# B&R Automation Studio project vibratorControlWithCurrentController (part 4)

#### brdkUpdate.fun - Exported functions and function blocks
```iecst
FUNCTION_BLOCK brdkUpdateCheck (*Reads the information from an update package.*) (*$GROUP=User,$CAT=User,$GROUPICON=User.png,$CATICON=User.png*)
	VAR_INPUT
		enable : BOOL := FALSE; (*Enables the function block.*)
		pFileDevice : UDINT := 0; (*String pointer for file device. Can be created with brdkFilelibrary.*)
	END_VAR
	VAR_OUTPUT
		updateFolderPath : STRING[255] := ''; (*Path of the update folder.*)
		pipFilePath : STRING[255] := ''; (*Path of the pipconfig.xml file.*)
		artransferFilePath : STRING[255] := ''; (*Filepath to "artransfer.br" file*)
		version : STRING[32] := ''; (*Update version number.*)
		id : STRING[255] := ''; (*Update configuration ID.*)
		artransferFileSize : UDINT := 0; (*Update file "artransfer.br" size in bytes.*)
		status : DINT := ERR_FUB_ENABLE_FALSE; (*Status of the function block.*)
	END_VAR
	VAR
		internal : brdk_update_check_internal_typ; (*Internal variables.*)
	END_VAR
END_FUNCTION_BLOCK

FUNCTION brdkUpdateCmpVersion : DINT (*Can compare two version strings. The version string must comply with Semantic Versioning x.x.x. $RETURN=result/error;1 : new > old- 0 : new = old : -1 new < old.*) (*$GROUP=User,$CAT=User,$GROUPICON=User.png,$CATICON=User.png*)
	VAR_INPUT
		pNewVersion : UDINT := 0; (*String pointer to new version.*)
		pOldVersion : UDINT := 0; (*String pointer to old version.*)
	END_VAR
END_FUNCTION

FUNCTION_BLOCK brdkUpdateDelete (*Deletes an update.*) (*$GROUP=User,$CAT=User,$GROUPICON=User.png,$CATICON=User.png*)
	VAR_INPUT
		enable : BOOL := FALSE; (*Enables the function block.*)
		pFileDevice : UDINT := 0; (*String pointer for file device. Can be created with brdkFilelibrary.*)
	END_VAR
	VAR_OUTPUT
		status : DINT := ERR_FUB_ENABLE_FALSE; (*Status of the function block.*)
	END_VAR
	VAR
		internal : brdk_update_delete_internal_typ; (*Internal variables.*)
	END_VAR
END_FUNCTION_BLOCK

FUNCTION_BLOCK brdkUpdateDistributeFTP (*Distributes an update package to a list of PLC's.*) (*$GROUP=User,$CAT=User,$GROUPICON=User.png,$CATICON=User.png*)
	VAR_INPUT
		enable : BOOL := FALSE; (*Enables the function block.*)
		pFileDevice : UDINT := 0; (*String pointer for file device. Can be created with brdkFilelibrary.*)
		client : ARRAY[0..BRDK_UPDATE_MAX_FTP_CLIENTS] OF brdk_update_dist_ftp_client_typ; (*List of FTP clients that will receive the update.*)
		cmd : brdk_update_dist_ftp_cmd_typ; (*Commands.*)
	END_VAR
	VAR_OUTPUT
		status : DINT := ERR_FUB_ENABLE_FALSE; (*Status of the function block.*)
		ready : BOOL := FALSE; (*Function block ready.*)
		version : STRING[32] := ''; (*Update version number.*)
		id : STRING[255] := ''; (*Update configuration ID.*)
		artransferFileSize : UDINT := 0; (*Update file "artransfer.br" size in bytes.*)
		updatePackagesSent : USINT := 0; (*Amount of update packages sent*)
	END_VAR
	VAR
		internal : brdk_update_dist_ftp_int_typ; (*Internal variables.*)
	END_VAR
END_FUNCTION_BLOCK

FUNCTION_BLOCK brdkUpdateManager (*Manages updates.*) (*$GROUP=User,$CAT=User,$GROUPICON=User.png,$CATICON=User.png*)
	VAR_INPUT
		enable : BOOL := FALSE; (*Enables the function block.*)
		pFileDevice : UDINT := 0; (*String pointer for file device. Can be created with brdkFilelibrary.*)
		cmd : brdk_update_manager_cmd_typ; (*Commands.*)
	END_VAR
	VAR_OUTPUT
		running : brdk_update_manager_run_info_typ; (*Running information.*)
		update : brdk_update_manager_upd_info_typ; (*Update information.*)
		ready : BOOL := FALSE; (*Function block ready.*)
		status : DINT := ERR_FUB_ENABLE_FALSE; (*Status of the function block.*)
	END_VAR
	VAR
		internal : brdk_update_manager_internal_typ; (*Internal variables.*)
	END_VAR
END_FUNCTION_BLOCK
```

#### brdkUpdateCheck.c - Reads the information from an update package.
```c
#include <brdkUpdate_func.h>

void brdkUpdateCheck(struct brdkUpdateCheck* inst) {
	brdk_update_check_internal_typ* this = (brdk_update_check_internal_typ*)&inst->internal;

	if(!inst->enable) {
		inst->status = ERR_FUB_ENABLE_FALSE;
		this->state = 0;
	}
	else {

		switch(this->state) {

			case 0: /* check that all pointers are set */
				inst->status = ERR_FUB_BUSY;
				if(inst->pFileDevice != 0) {
					this->simulation = DiagCpuIsARsim();
					this->brdkFileRead_0.enable 		= false;
					brdkFileRead(&this->brdkFileRead_0);
					this->brdkFileRead_0.enable 		= true;
					this->brdkFileRead_0.pFileDevice 	= inst->pFileDevice;
					this->brdkFileRead_0.pFileName 		= (unsigned long)&BRDK_UPDATE_DEFAULT_FILE_NAME;
					this->brdkFileRead_0.pData 			= (unsigned long)&this->buffer;
					this->brdkFileRead_0.dataLength 	= sizeof(this->buffer);
					this->state 						= 10;
				}
				else {
					inst->status 	= BRDK_UPDATE_POINTER_ERROR;
					this->state 	= 999;
				}
				break;

			case 10: /* wait for file to be read */
				brdkFileRead(&this->brdkFileRead_0);
				switch(this->brdkFileRead_0.status) {

					case ERR_OK:
						/* find Path= */
						if(!brdkStrSubStrSearch((unsigned long)&inst->pipFilePath,(unsigned long)&this->buffer,(unsigned long)&"Path",(unsigned long)&"\"",2,true)) {
							inst->status = BRDK_UPDATE_PIP_FILE_ERROR;
							this->state = 999;
						}
						else {
							this->position = brdkStrSearch((unsigned long)&inst->pipFilePath, (unsigned long)&"/");
							if(this->position < 0) {
								inst->status = BRDK_UPDATE_PIP_FILE_ERROR;
								this->state = 999;
							}
							else {
								brdkStrMemClear((unsigned long)&inst->updateFolderPath,sizeof(inst->updateFolderPath));
								brdkStrMemCpy((unsigned long)&inst->updateFolderPath, (unsigned long)&inst->pipFilePath, this->position);
								if(!this->simulation) {
									this->ArProjectGetPackageInfo_0.Execute = false;
									ArProjectGetPackageInfo(&this->ArProjectGetPackageInfo_0);
									brdkStrCpy((unsigned long)&this->ArProjectGetPackageInfo_0.DeviceName, inst->pFileDevice);
									brdkStrCpy((unsigned long)&this->ArProjectGetPackageInfo_0.FilePath, (unsigned long)&inst->pipFilePath);
									this->ArProjectGetPackageInfo_0.Execute = true;
									this->state 							= 20;
								}
								else {	/* ArProjectGetPackageInfo_0 does not work in simulation :-( we will just read the file our self ;-) */
									this->brdkFileRead_0.enable 		= false;
									brdkFileRead(&this->brdkFileRead_0);
									this->brdkFileRead_0.enable 		= true;
									this->brdkFileRead_0.pFileDevice 	= inst->pFileDevice;
									this->brdkFileRead_0.pFileName 		= (unsigned long)&inst->pipFilePath;
									this->brdkFileRead_0.pData 			= (unsigned long)&this->buffer;
									this->brdkFileRead_0.dataLength 	= sizeof(this->buffer);
									this->state 						= 30;
								}
							}
						}
						break;

					case ERR_FUB_BUSY:
						break;

					default:
						inst->status = this->brdkFileRead_0.status;
						break;
				}
				break;

			case 20: /* read update package info */
				ArProjectGetPackageInfo(&this->ArProjectGetPackageInfo_0);
				if(!this->ArProjectGetPackageInfo_0.Error) {
					if(this->ArProjectGetPackageInfo_0.Done) {
						brdkStrCpy((unsigned long)&inst->id,(unsigned long)&this->ArProjectGetPackageInfo_0.ConfigurationID);
						brdkStrCpy((unsigned long)&inst->version,(unsigned long)&this->ArProjectGetPackageInfo_0.ConfigurationVersion);

						this->FileInfo_0.enable = false;
						FileInfo(&this->FileInfo_0);
						this->FileInfo_0.enable = true;
						this->FileInfo_0.pDevice = inst->pFileDevice;
						brdkStrMemClear((unsigned long)&inst->artransferFilePath,sizeof(inst->artransferFilePath));
						brdkStrMemCpy((unsigned long)&inst->artransferFilePath,(unsigned long)&inst->updateFolderPath,sizeof(inst->updateFolderPath));
						brdkStrCat((unsigned long)&inst->artransferFilePath,(unsigned long)&BRDK_UPDATE_AR_TRANSFER_PATH);
						this->FileInfo_0.pName = (unsigned long)&inst->artransferFilePath;
						this->FileInfo_0.pInfo = (unsigned long)&this->updateFileInfo;
						this->state 	= 25;
					}
				}
				else {
					inst->status = this->ArProjectGetPackageInfo_0.StatusID;
				}
				break;

			case 25: /* Read file size of the binary update file "artransfer.br" */
				FileInfo(&this->FileInfo_0);
				switch(this->FileInfo_0.status){

					case ERR_OK:
						inst->artransferFileSize = this->updateFileInfo.size;
						inst->status = ERR_OK;
						this->state = 100;
						break;

					case ERR_FUB_BUSY:
						break;

					default:
						inst->status = this->FileInfo_0.status;
						break;

				}
				break;

			case 30: /* file open pipconfig.xml NB! only for simulation !!! */
				brdkFileRead(&this->brdkFileRead_0);
				switch(this->brdkFileRead_0.status) {

					case ERR_OK:
						/* find configuration ID e.g. <ConfigId>brdkUpdate_Config1</ConfigId> */
						if(!brdkStrSubStrSearch((unsigned long)&inst->id,(unsigned long)&this->buffer,(unsigned long)&"ConfigId",(unsigned long)&"<",1,true)) {
							inst->status = BRDK_UPDATE_PIP_FILE_ERROR;
							this->state = 999;
						}
						else {
							/* find configuration version e.g. <ConfigVersion>1.0.1</ConfigVersion> */
							if(!brdkStrSubStrSearch((unsigned long)&inst->version,(unsigned long)&this->buffer,(unsigned long)&"ConfigVersion",(unsigned long)&"<",1,true)) {
								inst->status = BRDK_UPDATE_PIP_FILE_ERROR;
								this->state = 999;
							}
							else {
								inst->status 	= ERR_OK;
								this->state 	= 100;
							}
						}
						break;

					case ERR_FUB_BUSY:
						break;

					default:
						inst->status = this->brdkFileRead_0.status;
						break;
				}
				break;

			case 100:
				break;

		}
	}
}
```

#### brdkUpdateCmpVersion.c - Can compare two version strings. The version string must comply with Semantic Versioning x.x.x
```c
#include <brdkUpdate_func.h>

signed long brdkUpdateCmpVersion(unsigned long pNewVersion, unsigned long pOldVersion) {
	unsigned long newIdx = 0, oldIdx = 0, newVal = 0, oldVal = 0, cnt = 0;
	char noZero;
	if(pNewVersion != 0 && pOldVersion != 0) {
		while(cnt < 3) {
			noZero = 0;
			while(((char*)pNewVersion)[newIdx] != 46 && ((char*)pNewVersion)[newIdx] != 0) {	/* look for a . */
				if((((char*)pNewVersion)[newIdx]) > 48) noZero = true;	/* make sure that first char is not a 0 */
				if(noZero) newVal += ((char*)pNewVersion)[newIdx];
				newIdx++;
			}
			newIdx++;
			noZero = 0;
			while(((char*)pOldVersion)[oldIdx] != 46 && ((char*)pOldVersion)[oldIdx] != 0) {	/* look for a . */
				if((((char*)pOldVersion)[oldIdx]) > 48) noZero = true;	/* make sure that first char is not a 0 */
				if(noZero) oldVal += ((char*)pOldVersion)[oldIdx];
				oldIdx++;
			}
			oldIdx++;
			if(newVal > oldVal) return 1;
			else if(newVal < oldVal) return -1;
			newVal = oldVal = 0;
			cnt++;
		}
	}
	else return BRDK_UPDATE_POINTER_ERROR;
	return 0;
}
```

#### brdkUpdateDelete.c - Deletes an update.
```c
#include <brdkUpdate_func.h>

void brdkUpdateDelete(struct brdkUpdateDelete* inst) {
	brdk_update_delete_internal_typ* this = (brdk_update_delete_internal_typ*)&inst->internal;

	if(!inst->enable) {
		inst->status = ERR_FUB_ENABLE_FALSE;
		this->state = 0;
	}
	else {

		switch(this->state) {

			case 0: /* check that all pointers are set */
				inst->status = ERR_FUB_BUSY;
				if(inst->pFileDevice != 0) {
					inst->status 						= ERR_FUB_BUSY;
					this->brdkUpdateCheck_0.enable 		= false;
					brdkUpdateCheck(&this->brdkUpdateCheck_0);
					this->brdkUpdateCheck_0.enable 		= true;
					this->brdkUpdateCheck_0.pFileDevice = inst->pFileDevice;
					this->state 						= 10;
				}
				else {
					inst->status 	= BRDK_UPDATE_POINTER_ERROR;
					this->state 	= 999;
				}
				break;

			case 10:
				brdkUpdateCheck(&this->brdkUpdateCheck_0);
				switch(this->brdkUpdateCheck_0.status) {

					case ERR_OK:
						this->DirDeleteEx_0.enable = false;
						DirDeleteEx(&this->DirDeleteEx_0);
						this->DirDeleteEx_0.enable 	= true;
						this->DirDeleteEx_0.pDevice = inst->pFileDevice;
						this->DirDeleteEx_0.pName 	= (unsigned long)&this->brdkUpdateCheck_0.updateFolderPath;
						this->state 				= 20;
						break;

					case ERR_FUB_BUSY:
						break;

					default:
						inst->status = this->brdkUpdateCheck_0.status;
						break;
				}
				break;

			case 20: /* delete update folder */
				DirDeleteEx(&this->DirDeleteEx_0);
				switch(this->DirDeleteEx_0.status) {

					case ERR_OK:
						this->FileDelete_0.enable = false;
						FileDelete(&this->FileDelete_0);
						this->FileDelete_0.enable 	= true;
						this->FileDelete_0.pDevice 	= inst->pFileDevice;
						this->FileDelete_0.pName 	= (unsigned long)&BRDK_UPDATE_DEFAULT_FILE_NAME;
						this->state 				= 30;
						break;

					case ERR_FUB_BUSY:
						break;

					default:
						inst->status = this->DirDeleteEx_0.status;
						break;

				}
				break;

			case 30: /* delete update file */
				FileDelete(&this->FileDelete_0);
				switch(this->FileDelete_0.status) {

					case ERR_OK:
						inst->status 	= ERR_OK;
						this->state 	= 40;
						break;

					case ERR_FUB_BUSY:
						break;

					default:
						inst->status = this->FileDelete_0.status;
						break;

				}
				break;

			case 40: /* done */
				break;

		}
	}
}
```

#### brdkUpdateDistributeFTP.c - Distributes an update package to a list of PLC's via FTP
```c
#include <brdkUpdate_func.h>

void brdkUpdateDistributeFTP(struct brdkUpdateDistributeFTP* inst) {
	brdk_update_dist_ftp_int_typ* this = (brdk_update_dist_ftp_int_typ*) &inst->internal;

	if(!inst->enable) {
		inst->status = ERR_FUB_ENABLE_FALSE;
		this->state = 0;
	}
	else {
		switch(this->state) {

			case 0: /* check that the file device pointer is set */
				if(inst->pFileDevice != 0) {
					inst->status = ERR_OK;
					inst->ready = true;
					this->state = 100;
				}
				else {
					inst->status 	= BRDK_UPDATE_POINTER_ERROR;
					this->state 	= 999;
				}
				break;

			case 100: /* wait for command */
				if(inst->cmd.distributeUpdate || inst->cmd.checkUpdate) {
					inst->ready 						= false;
					inst->status 						= ERR_FUB_BUSY;
					this->brdkUpdateCheck_0.enable 		= false;
					brdkUpdateCheck(&this->brdkUpdateCheck_0);
					this->brdkUpdateCheck_0.enable 		= true;
					this->brdkUpdateCheck_0.pFileDevice	= inst->pFileDevice;
					this->state 						= 110;
				}
				else if(inst->cmd.deleteUpdate) {
					inst->cmd.deleteUpdate 					= false;
					this->brdkUpdateDelete_0.enable			= false;
					brdkUpdateDelete(&this->brdkUpdateDelete_0);
					this->brdkUpdateDelete_0.enable 		= true;
					this->brdkUpdateDelete_0.pFileDevice 	= inst->pFileDevice;
					this->state 							= 200;
				}
				break;

			case 110: /* wait for update to be read */
				brdkUpdateCheck(&this->brdkUpdateCheck_0);
				switch(this->brdkUpdateCheck_0.status) {

					case ERR_OK:
						brdkStrCpy((unsigned long)&inst->id,(unsigned long)&this->brdkUpdateCheck_0.id);
						brdkStrCpy((unsigned long)&inst->version,(unsigned long)&this->brdkUpdateCheck_0.version);
						inst->artransferFileSize = this->brdkUpdateCheck_0.artransferFileSize;
						if(inst->cmd.checkUpdate) {
							inst->cmd.checkUpdate	= false;
							inst->status 			= ERR_OK;
							inst->ready 			= true;
							this->state 			= 100;
						}
						else if(inst->cmd.distributeUpdate) {
							inst->cmd.distributeUpdate = false;
							this->cIdx = 0;						/* reset client idx */
							inst->updatePackagesSent = 0;		/* reset packages sent */
							if(!brdkStrIsEmpty((unsigned long)&inst->client[this->cIdx].pIPAddress)) {
								brdkStrCpy((unsigned long)&this->paramStr,(unsigned long)&"/PROTOCOL=ftp");
								brdkStrCat((unsigned long)&this->paramStr,(unsigned long)&" /SIP=");
								brdkStrCat((unsigned long)&this->paramStr,inst->client[this->cIdx].pIPAddress);
								if(!brdkStrIsEmpty((unsigned long)&inst->client[this->cIdx].pUser)) {
									brdkStrCat((unsigned long)&this->paramStr,(unsigned long)&" /USER=");
									brdkStrCat((unsigned long)&this->paramStr,inst->client[this->cIdx].pUser);
									if(!brdkStrIsEmpty((unsigned long)&inst->client[this->cIdx].pPassword)) {
										brdkStrCat((unsigned long)&this->paramStr,(unsigned long)&" /PASSWORD=");
										brdkStrCat((unsigned long)&this->paramStr,inst->client[this->cIdx].pPassword);
									}
								}
								this->DevLink_0.enable = false;
								DevLink(&this->DevLink_0);
								this->DevLink_0.enable 	= true;
								this->DevLink_0.pDevice = (unsigned long)&BRDK_UPDATE_FTP_DEVICE_NAME;
								this->DevLink_0.pParam 	= (unsigned long)&this->paramStr;
								this->state 			= 120;
							}
						}
						break;

					case ERR_FUB_BUSY:
						break;

					default:
						inst->status = this->brdkUpdateCheck_0.status;
						if(inst->cmd.errorReset) {
							inst->cmd.errorReset 		= false;
							inst->cmd.distributeUpdate 	= false;
							inst->cmd.checkUpdate 		= false;
							inst->status 				= ERR_OK;
							inst->ready 				= true;
							this->state 				= 100;
						}
						break;
				}
				break;

			case 120: /* create dev link for FTP */
				DevLink(&this->DevLink_0);
				switch(this->DevLink_0.status) {

					case ERR_OK:
						this->DirCopy_0.enable 		= false;
						DirCopy(&this->DirCopy_0);
						this->DirCopy_0.enable 		= true;
						this->DirCopy_0.pSrcDev 	= inst->pFileDevice;
						this->DirCopy_0.pSrcDir 	= (unsigned long)&this->brdkUpdateCheck_0.updateFolderPath;
						this->DirCopy_0.pDestDev 	= this->DevLink_0.pDevice;
						this->DirCopy_0.pDestDir 	= 0;
						this->DirCopy_0.option 		= fiOVERWRITE;
						this->state 				= 130;
						break;

					case ERR_FUB_BUSY:
						break;

					default:
						inst->status 				= this->DevLink_0.status;
						if(inst->cmd.errorReset) {
							inst->cmd.errorReset 	= false;
							inst->status 			= ERR_OK;
							inst->ready 			= true;
							this->state 			= 100;
						}
						break;

				}
				break;

			case 130: /* copy update folder to ftp server */
				DirCopy(&this->DirCopy_0);
				switch(this->DirCopy_0.status) {

					case ERR_OK:
						this->FileCopy_0.enable 	= false;
						FileCopy(&this->FileCopy_0);
						this->FileCopy_0.enable 	= true;
						this->FileCopy_0.pSrcDev 	= this->DirCopy_0.pSrcDev;
						this->FileCopy_0.pSrc 		= (unsigned long)&BRDK_UPDATE_DEFAULT_FILE_NAME;
						this->FileCopy_0.pDestDev 	= this->DirCopy_0.pDestDev;
						this->FileCopy_0.pDest 		= this->FileCopy_0.pSrc;
						this->FileCopy_0.option 	= fiOVERWRITE;
						this->state 				= 140;
						break;

					case ERR_FUB_BUSY:
						break;

					default:
						inst->status 				= this->DirCopy_0.status;
						if(inst->cmd.errorReset) {
							inst->cmd.errorReset 	= false;
							inst->status 			= ERR_OK;
							inst->ready 			= true;
							this->state 			= 100;
						}
						break;

				}
				break;

			case 140: /* copy file */
				FileCopy(&this->FileCopy_0);
				switch(this->FileCopy_0.status) {

					case ERR_OK:
						this->DevUnlink_0.enable 	= false;
						DevUnlink(&this->DevUnlink_0);
						this->DevUnlink_0.enable 	= true;
						this->DevUnlink_0.handle 	= this->DevLink_0.handle;
						this->state 				= 150;
						break;

					case ERR_FUB_BUSY:
						break;

					default:
						inst->status 				= this->FileCopy_0.status;
						if(inst->cmd.errorReset) {
							inst->cmd.errorReset 	= false;
							inst->status 			= ERR_OK;
							inst->ready 			= true;
							this->state 			= 100;
						}
						break;

				}
				break;

			case 150: /* unlink file device */
				DevUnlink(&this->DevUnlink_0);
				switch(this->DevUnlink_0.status) {

					case ERR_OK:
						this->cIdx++;						/* reset client idx */
						inst->updatePackagesSent++;			/* Amount of packages sent	*/
						if(this->cIdx < BRDK_UPDATE_MAX_FTP_CLIENTS) {
							if(!brdkStrIsEmpty((unsigned long)&inst->client[this->cIdx].pIPAddress)) {
								brdkStrCpy((unsigned long)&this->paramStr,(unsigned long)&"/PROTOCOL=ftp");
								brdkStrCat((unsigned long)&this->paramStr,(unsigned long)&" /SIP=");
								brdkStrCat((unsigned long)&this->paramStr,inst->client[this->cIdx].pIPAddress);
								if(!brdkStrIsEmpty((unsigned long)&inst->client[this->cIdx].pUser)) {
									brdkStrCat((unsigned long)&this->paramStr,(unsigned long)&" /USER=");
									brdkStrCat((unsigned long)&this->paramStr,inst->client[this->cIdx].pUser);
									if(!brdkStrIsEmpty((unsigned long)&inst->client[this->cIdx].pPassword)) {
										brdkStrCat((unsigned long)&this->paramStr,(unsigned long)&" /PASSWORD=");
										brdkStrCat((unsigned long)&this->paramStr,inst->client[this->cIdx].pPassword);
									}
								}
								this->DevLink_0.enable = false;
								DevLink(&this->DevLink_0);
								this->DevLink_0.enable 	= true;
								this->DevLink_0.pDevice = (unsigned long)&BRDK_UPDATE_FTP_DEVICE_NAME;
								this->DevLink_0.pParam 	= (unsigned long)&this->paramStr;
								this->state 			= 120;
							}
							else {
								inst->status = ERR_OK;
								inst->ready = true;
								this->state = 100;
							}
						}
						else {
							inst->status = ERR_OK;
							inst->ready = true;
							this->state = 100;
						}
						break;

					case ERR_FUB_BUSY:
						break;

					default:
						inst->status 				= this->DevUnlink_0.status;
						if(inst->cmd.errorReset) {
							inst->cmd.errorReset 	= false;
							inst->status 			= ERR_OK;
							inst->ready 			= true;
							this->state 			= 100;
						}
						break;

				}
				break;

			case 200: /* delete update folder */
				brdkUpdateDelete(&this->brdkUpdateDelete_0);
				switch(this->brdkUpdateDelete_0.status) {

					case ERR_OK:
						inst->id[0] 		= 0;
						inst->version[0] 	= 0;
						inst->status 		= BRDK_UPDATE_NOT_FOUND;
						inst->status 		= ERR_OK;
						inst->ready 		= true;
						this->state 		= 100;
						break;

					case ERR_FUB_BUSY:
						break;

					default:
						inst->status = this->brdkUpdateDelete_0.status;
						if(inst->cmd.errorReset) {
							inst->cmd.errorReset = false;
							inst->status = ERR_OK;
							inst->ready = true;
							this->state = 100;
						}
						break;

				}
				break;

		}

	}
}
```

#### brdkUpdateManager.c - Manages updates.
```c
#include <brdkUpdate_func.h>

void brdkUpdateManager(struct brdkUpdateManager* inst) {
	brdk_update_manager_internal_typ* this = (brdk_update_manager_internal_typ*)&inst->internal;

	if(!inst->enable) {
		inst->status = ERR_FUB_ENABLE_FALSE;
		this->state = 0;
	}
	else {
		switch(this->state) {

			case 0: /* check that the file device pointer is set */
				inst->status = ERR_FUB_BUSY;
				if(inst->pFileDevice != 0) {
					this->ArProjectGetInfo_0.Execute = false;
					ArProjectGetInfo(&this->ArProjectGetInfo_0);
					this->ArProjectGetInfo_0.Execute = true;
					this->state = 10;
				}
				else {
					inst->status 	= BRDK_UPDATE_POINTER_ERROR;
					this->state 	= 999;
				}
				break;

			case 10: /* read the running id and version */
				ArProjectGetInfo(&this->ArProjectGetInfo_0);
				if(!this->ArProjectGetInfo_0.Error) {
					if(this->ArProjectGetInfo_0.Done) {
						brdkStrCpy((unsigned long)&inst->running.id,(unsigned long)&this->ArProjectGetInfo_0.ConfigurationID);
						brdkStrCpy((unsigned long)&inst->running.version,(unsigned long)&this->ArProjectGetInfo_0.ConfigurationVersion);
						inst->status = ERR_OK;
						inst->ready = true;
						this->state = 100;
					}
				}
				else {
					inst->status = this->ArProjectGetInfo_0.StatusID;
					if(inst->cmd.errorReset) {
						inst->cmd.errorReset = false;
						inst->status = ERR_OK;
						inst->ready = true;
						this->state = 100;
					}
				}
				break;

			case 100: /* check for commands */
				if(inst->cmd.checkForUpdate || inst->cmd.update || inst->cmd.updateReboot) {
					inst->ready 						= false;
					inst->status 						= ERR_FUB_BUSY;
					this->brdkUpdateCheck_0.enable 		= false;
					brdkUpdateCheck(&this->brdkUpdateCheck_0);
					this->brdkUpdateCheck_0.enable 		= true;
					this->brdkUpdateCheck_0.pFileDevice = inst->pFileDevice;
					this->state 						= 110;
				}
				else if(inst->cmd.deleteUpdate) {
					inst->cmd.deleteUpdate 					= false;
					this->brdkUpdateDelete_0.enable			= false;
					brdkUpdateDelete(&this->brdkUpdateDelete_0);
					this->brdkUpdateDelete_0.enable 		= true;
					this->brdkUpdateDelete_0.pFileDevice 	= inst->pFileDevice;
					this->state 							= 200;
				}
				break;

			case 110: /* wait for update to be read */
				brdkUpdateCheck(&this->brdkUpdateCheck_0);
				switch(this->brdkUpdateCheck_0.status) {

					case ERR_OK:
						if(inst->cmd.checkForUpdate) {
							inst->cmd.checkForUpdate				= false;
							brdkStrCpy((unsigned long)&inst->update.id,(unsigned long)&this->brdkUpdateCheck_0.id);
							brdkStrCpy((unsigned long)&inst->update.version,(unsigned long)&this->brdkUpdateCheck_0.version);
							inst->update.artransferFileSize = this->brdkUpdateCheck_0.artransferFileSize;
							inst->update.status = BRDK_UPDATE_NOT_FOUND;
							if(brdkStrCmp((unsigned long)&inst->update.id,(unsigned long)&inst->running.id) != 0) inst->update.status = BRDK_UPDATE_NO_ID_MATCH;
							this->versionCmp = brdkUpdateCmpVersion((unsigned long)&inst->update.version,(unsigned long)&inst->running.version);
							if(inst->update.status != BRDK_UPDATE_NO_ID_MATCH) {
								if(this->versionCmp > 0) inst->update.status = BRDK_UPDATE_VERSION_NEW_GREATER;
								else if(this->versionCmp < 0) inst->update.status = BRDK_UPDATE_VERSION_NEW_SMALLER;
								else inst->update.status = BRDK_UPDATE_VERSIONS_EQUAL;
							}
							inst->status 	= ERR_OK;
							inst->ready 	= true;
							this->state 	= 100;
						}
						else if(inst->cmd.update || inst->cmd.updateReboot) {
							inst->cmd.update 						= false;
							this->ArProjectInstallPackage_0.Execute = false;
							ArProjectInstallPackage(&this->ArProjectInstallPackage_0);
							this->ArProjectInstallPackage_0.Execute = true;
							brdkStrCpy((unsigned long)&this->ArProjectInstallPackage_0.DeviceName, inst->pFileDevice);
							brdkStrCpy((unsigned long)&this->ArProjectInstallPackage_0.FilePath, (unsigned long)&this->brdkUpdateCheck_0.pipFilePath);
							this->state 							= 300;
						}
						break;

					case ERR_FUB_BUSY:
						break;

					default:
						inst->status = this->brdkUpdateCheck_0.status;
						if(inst->cmd.errorReset) {
							inst->cmd.errorReset 		= false;
							inst->cmd.checkForUpdate 	= false;
							inst->cmd.update 			= false;
							inst->cmd.updateReboot		= false;
							inst->status 				= ERR_OK;
							inst->ready 				= true;
							this->state 				= 100;
						}
						break;
				}
				break;

			case 200: /* delete update folder */
				brdkUpdateDelete(&this->brdkUpdateDelete_0);
				switch(this->brdkUpdateDelete_0.status) {

					case ERR_OK:
						inst->update.id[0] 		= 0;
						inst->update.version[0] = 0;
						inst->update.status 	= BRDK_UPDATE_NOT_FOUND;
						inst->status 			= ERR_OK;
						inst->ready 			= true;
						this->state 			= 100;
						break;

					case ERR_FUB_BUSY:
						break;

					default:
						inst->status = this->brdkUpdateDelete_0.status;
						if(inst->cmd.errorReset) {
							inst->cmd.errorReset = false;
							inst->status = ERR_OK;
							inst->ready = true;
							this->state = 100;
						}
						break;

				}
				break;

			case 300: /* install update package */
				ArProjectInstallPackage(&this->ArProjectInstallPackage_0);
				if(!this->ArProjectInstallPackage_0.Error) {
					if(this->ArProjectInstallPackage_0.Done) {
						if(!inst->cmd.updateReboot) {
							inst->cmd.checkForUpdate 	= true;
							this->state 				= 0;
						}
						else {
							inst->cmd.updateReboot = false;
							SYSreset(true,1);	/* warm restart */
						}
					}
				}
				else {
					inst->status = this->ArProjectInstallPackage_0.StatusID;
					if(inst->cmd.errorReset) {
						inst->cmd.errorReset = false;
						inst->status = ERR_OK;
						inst->ready = true;
						this->state = 100;
					}
				}
				break;

			case 999: /* error state */
				if(inst->cmd.errorReset) {
					inst->cmd.errorReset 	= false;
					inst->cmd.updateReboot 	= false;
					inst->status 			= ERR_OK;
					inst->ready 			= true;
					this->state 			= 100;
				}
				break;

		}

	}
}
```

#### brdkUpdate_func.h - Common library header.
```c
#ifndef BRDK_UPDATE_FUNCS
#define BRDK_UPDATE_FUNCS 1

#include <brdkUpdate.h>
#include <bur/plctypes.h>

#ifdef __cplusplus
	extern "C"
	{
#endif

#ifdef __cplusplus
	};
#endif

#define false 0
#define true 1
#define NULL 0

#endif /* !BRDK_UPDATE_FUNCS */
```

- CHANGELOG - Change log. (not shown)

### Library Logical/Libraries/brdkFile (ANSIC, version 1.00.0) - File handling library. Makes it easy to handle file devices and to do file handling.
Depends on: AsIODiag, AsUSB, FileIO, brdkSTR

#### brdkFile.typ - Data types
```iecst
TYPE
	brdk_file_dev_handler_int_typ : 	STRUCT  (*Internal variables.*)
		fileState : UINT; (*State of the file device handler.*)
		driveState : UINT; (*State of the drive handler.*)
		DevLink_0 : DevLink; (*Device link.*)
		DevUnlink_0 : DevUnlink; (*Device unlink.*)
		DirInfo_0 : DirInfo; (*Directory create.*)
		drive : STRING[10]; (*Drive.*)
		deviceParam : STRING[BRDK_FILE_MAX_PATH_LEN]; (*Device parameter string.*)
		fileIdx : DINT; (*File index.*)
		activeHandles : ARRAY[0..BRDK_FILE_MAX_FILES_DEVICES]OF UDINT; (*Active handles.*)
		driveReady : BOOL; (*Drive ready to use.*)
		oldUseUSB : BOOL; (*Holds the old command.*)
		usbOK : BOOL; (*USB drive present and ready to use.*)
		brdkFileCreateSubFolders_0 : brdkFileCreateSubFolders; (*Create sub folders.*)
		UsbNodeListGet_0 : UsbNodeListGet; (*Get list of USB nodes.*)
		UsbNodeGet_0 : UsbNodeGet; (*Get USB node.*)
		nodeId : ARRAY[0..BRDK_FILE_MAX_USB_NODES]OF UDINT; (*Node id buffer list.*)
		nodeIdx : USINT; (*Node id index.*)
		usbNode : usbNode_typ; (*Node info.*)
		oldUSBok : BOOL; (*Holds the old status.*)
		oldNodeId : UDINT; (*Holds the old node id.*)
		usbHandles : ARRAY[0..BRDK_FILE_MAX_FILES_DEVICES]OF DINT := [10(-1)]; (*Hold the USB handles.*)
	END_STRUCT;
	brdk_file_dev_handler_sim_typ : 	STRUCT  (*Simulation options.*)
		pcRootFolder : STRING[BRDK_FILE_MAX_PATH_LEN] := 'plcRoot'; (*Path on the PC that will simulate the root of the controller. Default plcRoot -> C:\plcRoot\*)
		pcUSBDrive : brdk_file_drive_typ := D_DRIVE; (*Drive letter of the PC's USB. Default D:\.*)
		pcHDDrive : brdk_file_drive_typ := C_DRIVE; (*Drive letter of the PC's HD. Default C:\.*)
	END_STRUCT;
	brdk_file_dev_handler_setup_typ : 	STRUCT  (*Setup options.*)
		plcDrive : brdk_file_drive_typ := C_DRIVE; (*Drive letter of the controller flash. Default C:\.*)
		usbOverrule : BOOL := FALSE; (*Inserted USB stick will overrule internal flash if the USB stick is present.*)
		fileDevices : ARRAY[0..BRDK_FILE_MAX_FILES_DEVICES]OF brdk_file_file_devices_typ; (*File devices. Default CONFIG and RECEIPES with config and recipes folder.*)
		keepHDAlive : BOOL := FALSE; (*Keeps the HD alive when the USB is inserted.*)
	END_STRUCT;
	brdk_file_drive_typ :
		( (*Drive selection. Default C:\.*)
		C_DRIVE := 0, (*C:\*)
		D_DRIVE := 1, (*D:\*)
		E_DRIVE := 2, (*E:\*)
		F_DRIVE := 3, (*F:\*)
		G_DRIVE := 4 (*G:\*)
		) := C_DRIVE;
	brdk_file_file_devices_typ : 	STRUCT  (*File devices setup.*)
		name : STRING[BRFK_FILE_MAX_FILE_DEVICE_LEN]; (*Name of the file device to be used as input for file functions.*)
		path : STRING[BRDK_FILE_MAX_PATH_LEN]; (*Folder path for the file device. Only the folders must be entered the drive is setup in the setup options. E.g. config.*)
	END_STRUCT;
	brdk_file_create_subfold_int_typ : 	STRUCT  (*Internal variables.*)
		state : DINT; (*State of the function block.*)
		DirCreate_0 : DirCreate; (*Directory create.*)
		tmpPath : STRING[BRDK_FILE_MAX_PATH_LEN]; (*Temp path string.*)
		pathPos : DINT; (*Path position.*)
		tmpPathPos : DINT; (*Tmp path position.*)
		tmpLen : DINT; (*Temp length.*)
	END_STRUCT;
	brdk_file_read_internal_typ : 	STRUCT  (*Internal variables.*)
		state : DINT; (*State of the function block.*)
		FileOpen_0 : FileOpen; (*File open.*)
		FileClose_0 : FileClose; (*File close.*)
		FileRead_0 : FileRead; (*File read.*)
	END_STRUCT;
	brdk_file_write_internal_typ : 	STRUCT  (*Internal variables.*)
		state : DINT; (*State of the function block.*)
		FileOpen_0 : FileOpen; (*File open.*)
		FileCreate_0 : FileCreate; (*File create.*)
		FileClose_0 : FileClose; (*File close.*)
		FileDelete_0 : FileDelete; (*File delete.*)
		FileWrite_0 : FileWrite; (*File write.*)
	END_STRUCT;
	brdk_file_file_device_status_typ : 	STRUCT  (*Status of the file devices.*)
		readyHD : BOOL := FALSE; (*Indicates that the HD drive is ready.*)
		readyUSB : BOOL := FALSE; (*Indicates that the USB drive is ready.*)
	END_STRUCT;
END_TYPE
```

#### brdkFile.var - Constants
```iecst
VAR CONSTANT
	BRDK_FILE_MAX_USB_NODES : USINT := 5; (*Maximum number of connected USB nodes. (5 means 6)*)
	BRDK_FILE_MAX_FILES_DEVICES : USINT := 9; (*Maximum numbers of file devices. (9 means 10)*)
	BRDK_FILE_MAX_PATH_LEN : UINT := 200; (*Maximum length of a path.*)
	BRFK_FILE_MAX_FILE_DEVICE_LEN : UINT := 50; (*Maximum length of file device names.*)
END_VAR
```

#### brdkFile.fun - Functions and function blocks
```iecst
FUNCTION_BLOCK brdkFileDeviceHandler (*Easy file device handler. This function block makes file device handling easy. The idea of the function block is that you only need to create one file device name that can be used for both internal and usb flash.*) (*$GROUP=User,$CAT=User,$GROUPICON=User.png,$CATICON=User.png*)
	VAR_INPUT
		enable : BOOL; (*Enables the function block.*)
		setup : brdk_file_dev_handler_setup_typ; (*Setup options.*)
		simulation : brdk_file_dev_handler_sim_typ; (*Simulation options.*)
		useUSB : BOOL; (*Stores on the USB if it is possible. Can be auto selected in the setup options.*)
	END_VAR
	VAR_OUTPUT
		availableDevices : ARRAY[0..BRDK_FILE_MAX_FILES_DEVICES] OF STRING[BRFK_FILE_MAX_FILE_DEVICE_LEN]; (*List of available file devices.*)
		ready : BOOL; (*Means that all file devices have been created and are ready to use.*)
		description : STRING[200]; (*Status description.*)
		status : UINT; (*Status of FileIO function blocks.*)
		fileDeviceStatus : ARRAY[0..BRDK_FILE_MAX_FILES_DEVICES] OF brdk_file_file_device_status_typ; (*Status of the file devices.*)
	END_VAR
	VAR
		internal : brdk_file_dev_handler_int_typ; (*Internal variables.*)
	END_VAR
END_FUNCTION_BLOCK

FUNCTION_BLOCK brdkFileCreateSubFolders (*Creates folders based on a path string.*) (*$GROUP=User,$CAT=User,$GROUPICON=User.png,$CATICON=User.png*)
	VAR_INPUT
		enable : BOOL; (*Enables the function block.*)
		path : STRING[BRDK_FILE_MAX_PATH_LEN]; (*Path of folder to be created. Use \ to seperate folders.*)
		fileDevice : STRING[BRFK_FILE_MAX_FILE_DEVICE_LEN]; (*File device name.*)
	END_VAR
	VAR_OUTPUT
		description : STRING[200]; (*Status description.*)
		done : BOOL; (*Function block done.*)
		status : UINT; (*Status of DirCreate function block.*)
	END_VAR
	VAR
		internal : brdk_file_create_subfold_int_typ; (*Internal variables.*)
	END_VAR
END_FUNCTION_BLOCK

FUNCTION_BLOCK brdkFileWrite (*Write data to a file.*) (*$GROUP=User,$CAT=User,$GROUPICON=User.png,$CATICON=User.png*)
	VAR_INPUT
		enable : BOOL; (*Enables the function block.*)
		pFileDevice : UDINT; (*String pointer to file device.*)
		pFileName : UDINT; (*String pointer to file name.*)
		pData : UDINT; (*Pointer to the data that must be written to the file.*)
		dataLength : UDINT; (*Length of the data that must be written. If 0 is specified \0 will end the data.*)
		overwrite : BOOL; (*Overwrite existing file. If not set the data will be appended to existing file.*)
	END_VAR
	VAR_OUTPUT
		status : UINT; (*Status of FileIO function blocks.*)
	END_VAR
	VAR
		internal : brdk_file_write_internal_typ; (*Internal variables.*)
	END_VAR
END_FUNCTION_BLOCK

FUNCTION_BLOCK brdkFileRead (*Read data from a file.*) (*$GROUP=User,$CAT=User,$GROUPICON=User.png,$CATICON=User.png*)
	VAR_INPUT
		enable : BOOL; (*Enables the function block.*)
		pFileDevice : UDINT; (*String pointer to file device.*)
		pFileName : UDINT; (*String pointer to file name.*)
		pData : UDINT; (*Pointer to the data where the data is read to.*)
		dataLength : UDINT; (*Length of the read data buffer.*)
	END_VAR
	VAR_OUTPUT
		status : UINT; (*Status of FileIO function blocks.*)
	END_VAR
	VAR
		internal : brdk_file_read_internal_typ; (*Internal variables.*)
	END_VAR
END_FUNCTION_BLOCK
```

#### brdkFileDeviceHandler.c - Easy file device handler.
```c
#include <brdkFile_func.h>

#define BR_TG_VENDOR_ID 1615
#define BR_TG_PRODUCT_ID 1001

void brdkFileDeviceHandler(struct brdkFileDeviceHandler* inst) {
	brdk_file_dev_handler_int_typ* this = (brdk_file_dev_handler_int_typ*)&inst->internal;		/* pointer to the internal structure */
	brdk_file_dev_handler_setup_typ* setup = (brdk_file_dev_handler_setup_typ*)&inst->setup;	/* pointer to the setup structure */
	brdk_file_dev_handler_sim_typ* sim = (brdk_file_dev_handler_sim_typ*)&inst->simulation;		/* pointer to the simulation structure */
	char tmpStr[200];

	if(inst->enable) {

		/* check weither the controller is beeing simulated and watch the usb status */
		if(!DiagCpuIsSimulated()) {
			if(!this->UsbNodeGet_0.enable) this->UsbNodeListGet_0.enable = true;
			this->UsbNodeListGet_0.pBuffer					= (unsigned long)&this->nodeId;
			this->UsbNodeListGet_0.bufferSize 				= sizeof(this->nodeId);
			this->UsbNodeListGet_0.filterInterfaceClass 	= asusb_CLASS_MASS_STORAGE;
			this->UsbNodeListGet_0.filterInterfaceSubClass 	= asusb_SUBCLASS_SCSI_COMMAND_SET;
			UsbNodeListGet(&this->UsbNodeListGet_0);
			if(this->UsbNodeListGet_0.status == asusbERR_USB_NOTFOUND) {
				this->nodeIdx = 0;
				this->usbOK = false;
			}

			this->UsbNodeGet_0.enable 		= true;
			this->UsbNodeGet_0.nodeId 		= this->nodeId[this->nodeIdx];
			this->UsbNodeGet_0.pBuffer 		= (unsigned long)&this->usbNode;
			this->UsbNodeGet_0.bufferSize 	= sizeof(this->usbNode);
			UsbNodeGet(&this->UsbNodeGet_0);
			if(this->UsbNodeGet_0.status == ERR_OK) {
				if(this->usbNode.vendorId == BR_TG_VENDOR_ID && this->usbNode.productId == BR_TG_PRODUCT_ID) {
					this->UsbNodeGet_0.enable 		= false;
					UsbNodeGet(&this->UsbNodeGet_0);
					this->nodeIdx++;
				}
				else this->usbOK = true;
			}
			else if(this->UsbNodeGet_0.status == asusbERR_USB_NOTFOUND) {
				this->UsbNodeListGet_0.enable = true;
				this->nodeIdx = 0;
				this->usbOK = false;
			}
			if(this->oldNodeId != this->UsbNodeGet_0.nodeId) this->usbOK = false;
			this->oldNodeId = this->UsbNodeGet_0.nodeId;
		}
		else {
			/* look for USB root folder */
			if(this->DirInfo_0.pDevice != 0) {
				this->DirInfo_0.enable 	= true;
				this->DirInfo_0.pPath 	= (unsigned long)"";
				DirInfo(&this->DirInfo_0);
				switch(this->DirInfo_0.status) {
					case 0: this->usbOK = true; break;
					case 20723: this->usbOK = false; break;
					default: break;
				}
			}
		}
		if(setup->usbOverrule) inst->useUSB = this->usbOK;	/* USB stick will overrule */
	}
	else {
		this->usbOK 					= false;
		this->nodeIdx 					= 0;
		this->DirInfo_0.enable 			= false;
		DirInfo(&this->DirInfo_0);
		this->UsbNodeGet_0.enable 		= false;
		UsbNodeGet(&this->UsbNodeGet_0);
		this->UsbNodeListGet_0.enable 	= false;
		UsbNodeListGet(&this->UsbNodeListGet_0);
	}

	/* drive handler */
	switch(this->driveState) {

		case 0:
			if(inst->enable) {
				if(!DiagCpuIsSimulated()) {	/* check if the controller is simulated */
					if((inst->useUSB && this->usbOK) || !inst->useUSB) {
						this->driveReady = true;
						if(!inst->useUSB) getDrive(setup->plcDrive,this->drive);
						else brdkStrCpy((unsigned long)this->drive,(unsigned long)this->usbNode.ifName);
						this->driveState = 499;
					}
				}
				else {
					this->DevLink_0.enable 	= true;
					this->DevLink_0.pDevice = (unsigned long)"INTUSB";
					this->DevLink_0.pParam 	= buildParameterString(getDrive(sim->pcUSBDrive,this->drive),(char*)&"",(char*)&this->deviceParam);
					this->driveState 		= 100;
				}
			}
			break;

		case 100:	/* create a file device for finding an attached usb flash */
			DevLink(&this->DevLink_0);
			if(this->DevLink_0.status != ERR_FUB_BUSY) {
				if(this->DevLink_0.status == ERR_OK || this->DevLink_0.status == fiERR_DEVICE_ALREADY_EXIST) {
					this->DirInfo_0.pDevice = this->DevLink_0.pDevice;
					this->DevLink_0.enable 	= false;
					DevLink(&this->DevLink_0);
					this->driveState 		= 110;
				}
				else {
					inst->status = this->DevLink_0.status;
					this->DevLink_0.enable 	= false;
					DevLink(&this->DevLink_0);
					brdkStrCpy((unsigned long)inst->description,(unsigned long)"error calling DevLink. Flip enable to reset fb.");
					this->driveState = 900;
				}
			}
			break;

		case 110:	/* wait for DirInfo to have been call once. Fb is call above */
			switch(this->DirInfo_0.status) {

				case 0: case 20723:
					if(!inst->useUSB) {
						getDrive(sim->pcHDDrive,this->drive);
						brdkStrCat((unsigned long)this->drive,(unsigned long)sim->pcRootFolder);
					}
					else getDrive(sim->pcUSBDrive,this->drive);
					this->driveState = 499;
					this->driveReady = true;
					break;

				case 65534: case 65535: break;

				default:
					inst->status 			= this->DirInfo_0.status;
					this->DirInfo_0.enable 	= false;
					DirInfo(&this->DirInfo_0);
					brdkStrCpy((unsigned long)inst->description,(unsigned long)"error calling DirInfo. Flip enable to reset fb.");
					this->driveReady = false;
					this->driveState = 900;
					break;

			}
			break;

		case 499:	/* waiting for file devices to be ready */
			if(!inst->enable) {
				this->driveReady = false;
				this->driveState = 900;
			}
			else if(inst->ready) this->driveState = 500;
			break;

		case 500:	/* check if USB status changes */
			if(!inst->enable) {
				this->driveReady = false;
				this->driveState = 900;
			}
			else if((this->oldUseUSB != inst->useUSB) || (inst->useUSB && (this->oldUSBok != this->usbOK))) {	/* usb must be used and the ok status has changed */
				this->driveReady = false;
				if(inst->useUSB && !this->usbOK) brdkStrCpy((unsigned long)inst->description,(unsigned long)"USB not ready. Turn off useUSB command.");
				else this->driveState = 510;
			}
			this->oldUseUSB = inst->useUSB;
			this->oldUSBok 	= this->usbOK;
			this->oldNodeId = this->UsbNodeGet_0.nodeId;
			break;

		case 510:	/* select the new drive */
			if(!DiagCpuIsSimulated()) {	/* check if the controller is simulated */
				if(!inst->useUSB) getDrive(setup->plcDrive,this->drive);
				else brdkStrCpy((unsigned long)this->drive,(unsigned long)this->usbNode.ifName);
			}
			else {
				if(!inst->useUSB) {
					getDrive(sim->pcHDDrive,this->drive);
					brdkStrCat((unsigned long)this->drive,(unsigned long)sim->pcRootFolder);
				}
				else getDrive(sim->pcUSBDrive,this->drive);
			}
			this->driveReady = true;
			this->driveState = 499;
			break;

		case 900:	/* error state */
			this->driveReady = false;
			if(!inst->enable) {
				inst->status 		= 0;
				this->driveState 	= 0;
			}
			break;

	}

	/* file device handler */
	switch(this->fileState) {

		case 0:	/* wait for a drive */
			if(inst->enable) {
				if(this->driveReady) {
					this->DevLink_0.enable 	= true;
					this->DevLink_0.pDevice = (this->usbOK) ? (unsigned long)"ROOT" : (unsigned long)"ROOT_USB";
					this->DevLink_0.pParam 	= buildParameterString((char*)&this->drive,(char*)&"",(char*)&this->deviceParam);
					this->fileState 		= 10;
				}
			}
			else {
				inst->ready = false;
			}
			break;

		case 10:
			brdkStrCpy((unsigned long)inst->description,(unsigned long)"creates a devlink for the drive root");
			DevLink(&this->DevLink_0);
			if(this->DevLink_0.status != ERR_FUB_BUSY) {
				if(this->DevLink_0.status == ERR_OK) {
					brdkStrCpy((unsigned long)inst->availableDevices[0],this->DevLink_0.pDevice);
					this->activeHandles[0] = this->DevLink_0.handle;
					this->DevLink_0.enable 	= false;
					DevLink(&this->DevLink_0);
					this->fileIdx = 0;
					if(setup->fileDevices[this->fileIdx].name[0] != 0) {
						brdkStrCpy((unsigned long)this->brdkFileCreateSubFolders_0.path,(unsigned long)setup->fileDevices[this->fileIdx].path);
						brdkStrCpy((unsigned long)this->brdkFileCreateSubFolders_0.fileDevice,this->DevLink_0.pDevice);
						this->brdkFileCreateSubFolders_0.enable = true;
						brdkFileCreateSubFolders(&this->brdkFileCreateSubFolders_0);
						this->fileState = 20;
					}
					else this->fileState = 100;
				}
				else if(this->DevLink_0.status == fiERR_DEVICE_ALREADY_EXIST) {
					if(this->DevLink_0.handle != 0) {
						inst->status = this->DevLink_0.status;
						this->DevLink_0.enable 	= false;
						DevLink(&this->DevLink_0);
						brdkStrCpy((unsigned long)inst->description,(unsigned long)"Device ");
						brdkStrCat((unsigned long)inst->description,this->DevLink_0.pDevice);
						brdkStrCat((unsigned long)inst->description,(unsigned long)" already exists. Reboot controller to kill the old device.");
						this->fileState = 900;
					}
					else {
						this->DevUnlink_0.enable = true;
						this->DevUnlink_0.handle = this->DevLink_0.handle;
						this->DevLink_0.enable 	= false;
						DevLink(&this->DevLink_0);
						this->fileState = 40;
					}
				}
				else {
					brdkStrCpy((unsigned long)inst->description,(unsigned long)"error calling DevLink. Flip enable to reset fb.");
					inst->status 			= this->DevLink_0.status;
					this->DevLink_0.enable 	= false;
					DevLink(&this->DevLink_0);
					this->fileState 		= 900;
				}
			}
			break;

		case 20:
			brdkStrCpy((unsigned long)inst->description,(unsigned long)"creates the needed folders");
			brdkFileCreateSubFolders(&this->brdkFileCreateSubFolders_0);
			if(this->brdkFileCreateSubFolders_0.done) {
				this->brdkFileCreateSubFolders_0.enable = false;
				brdkFileCreateSubFolders(&this->brdkFileCreateSubFolders_0);
				this->fileIdx++;
				if(setup->fileDevices[this->fileIdx].name[0] != 0 && setup->fileDevices[this->fileIdx].path[0] != 0) {
					this->brdkFileCreateSubFolders_0.enable = true;
					brdkStrCpy((unsigned long)this->brdkFileCreateSubFolders_0.path,(unsigned long)setup->fileDevices[this->fileIdx].path);
					brdkFileCreateSubFolders(&this->brdkFileCreateSubFolders_0);
				}
				else {
					this->fileIdx = 0;
					this->DevLink_0.enable 	= true;
					this->DevLink_0.pDevice = (unsigned long)setup->fileDevices[this->fileIdx].name;
					this->DevLink_0.pParam 	= buildParameterString((char*)&this->drive,(char*)&setup->fileDevices[this->fileIdx].path,(char*)&this->deviceParam);
					this->fileState = 30;
				}
			}
			else if(this->brdkFileCreateSubFolders_0.status == fiERR_FILE_DEVICE) {
				if(DiagCpuIsSimulated()) {
					this->DevUnlink_0.enable 	= true;
					this->DevUnlink_0.handle 	= this->activeHandles[0];
					this->activeHandles[0] 		= 0;
					DevUnlink(&this->DevUnlink_0);
					this->brdkFileCreateSubFolders_0.enable = false;
					brdkFileCreateSubFolders(&this->brdkFileCreateSubFolders_0);
					this->fileState 			= 200;
				}
				else {
					brdkStrCpy((unsigned long)inst->description,(unsigned long)"error calling brdkFileCreateSubFolders. Flip enable to reset fb.");
					inst->status 				= this->brdkFileCreateSubFolders_0.status;
					this->brdkFileCreateSubFolders_0.enable = false;
					brdkFileCreateSubFolders(&this->brdkFileCreateSubFolders_0);
					this->fileState 			= 900;
				}
			}
			else if(this->brdkFileCreateSubFolders_0.status != ERR_FUB_BUSY) brdkStrCpy((unsigned long)inst->description,(unsigned long)"error calling brdkFileCreateSubFolders. Check fb for error codes.");
			break;

		case 30:
			brdkStrCpy((unsigned long)inst->description,(unsigned long)"creates the needed file devices");
			DevLink(&this->DevLink_0);
			if(this->DevLink_0.status != ERR_FUB_BUSY) {
				if(this->DevLink_0.status == ERR_OK) {
					brdkStrCpy((unsigned long)inst->availableDevices[this->fileIdx+1],this->DevLink_0.pDevice);
					this->activeHandles[this->fileIdx+1] = this->DevLink_0.handle;
					this->DevLink_0.enable 	= false;
					DevLink(&this->DevLink_0);
					this->fileIdx++;
					if(setup->fileDevices[this->fileIdx].name[0] != 0 && setup->fileDevices[this->fileIdx].path[0] != 0) {
						this->DevLink_0.enable 	= true;
						this->DevLink_0.pDevice = (unsigned long)setup->fileDevices[this->fileIdx].name;
						this->DevLink_0.pParam 	= buildParameterString((char*)&this->drive,(char*)&setup->fileDevices[this->fileIdx].path,(char*)&this->deviceParam);
					}
					else {
						inst->ready = true;
						brdkStrCpy((unsigned long)inst->description,(unsigned long)"all file devices are ready to use");
						this->fileState = 100;
					}
				}
				else {
					brdkStrCpy((unsigned long)inst->description,(unsigned long)"error calling DevLink. Flip enable to reset fb.");
					inst->status 			= this->DevLink_0.status;
					this->DevLink_0.enable 	= false;
					DevLink(&this->DevLink_0);
					this->fileState 		= 900;
				}
			}
			break;

		case 40:
			DevUnlink(&this->DevUnlink_0);
			if(this->DevUnlink_0.status != ERR_FUB_BUSY) {
				if(this->DevUnlink_0.status == ERR_OK) {
					this->DevUnlink_0.enable = false;
					DevUnlink(&this->DevUnlink_0);
					this->DevLink_0.enable 	= true;
					this->DevLink_0.pDevice = (unsigned long)"ROOT";
					this->DevLink_0.pParam 	= buildParameterString((char*)&this->drive,(char*)&"",(char*)&this->deviceParam);
					this->fileState 		= 10;
				}
				else {
					brdkStrCpy((unsigned long)inst->description,(unsigned long)"error calling DevUnlink. Flip enable to reset fb.");
					inst->status 				= this->DevUnlink_0.status;
					this->DevUnlink_0.enable 	= false;
					DevUnlink(&this->DevUnlink_0);
					this->fileState 			= 900;
				}
			}
			break;

		case 100:	/* wait for interuption */
			if(!inst->enable) {
				inst->ready 	= false;
				this->fileState = 900;
			}
			if(!this->driveReady) {
				inst->ready = false;
				if(this->activeHandles[0] != 0) {
					this->fileIdx = 0;
					this->DevUnlink_0.handle 	= this->activeHandles[this->fileIdx];
					this->DevUnlink_0.enable 	= true;
					this->fileState 			= 110;
				}
				else this->fileState = 0;
			}
			break;

		case 110:	/* unlink file devices */
			DevUnlink(&this->DevUnlink_0);
			if(this->DevUnlink_0.status != ERR_FUB_BUSY) {
				if(this->DevUnlink_0.status == ERR_OK) {
					brdkStrCpy((unsigned long)inst->availableDevices[this->fileIdx],(unsigned long)"");
					this->activeHandles[this->fileIdx] = 0;
					this->fileIdx++;
					this->DevUnlink_0.enable = false;
					DevUnlink(&this->DevUnlink_0);
					if(this->activeHandles[this->fileIdx] != 0) {
						this->DevUnlink_0.enable = true;
						this->DevUnlink_0.handle = this->activeHandles[this->fileIdx];
					}
					else this->fileState = 0;
				}
				else {
					brdkStrCpy((unsigned long)inst->description,(unsigned long)"error calling DevUnlink. Flip enable to reset fb.");
					inst->status 				= this->DevUnlink_0.status;
					this->DevUnlink_0.enable 	= false;
					DevUnlink(&this->DevUnlink_0);
					this->fileState 			= 900;
				}
			}
			break;

		case 200:
			DevUnlink(&this->DevUnlink_0);
			if(this->DevUnlink_0.status != ERR_FUB_BUSY) {
				if(this->DevUnlink_0.status == ERR_OK) {
					this->DevUnlink_0.enable = false;
					DevUnlink(&this->DevUnlink_0);
					this->DevLink_0.enable 	= true;
					this->DevLink_0.pDevice = (unsigned long)"tmpRoot";
					this->DevLink_0.pParam 	= buildParameterString(getDrive(sim->pcHDDrive,tmpStr),(char*)&"",(char*)&this->deviceParam);
					this->fileState 		= 210;
				}
				else {
					brdkStrCpy((unsigned long)inst->description,(unsigned long)"error calling DevUnlink. Flip enable to reset fb.");
					inst->status 				= this->DevUnlink_0.status;
					this->DevUnlink_0.enable 	= false;
					DevUnlink(&this->DevUnlink_0);
					this->fileState 			= 900;
				}
			}
			break;

		case 210:
			brdkStrCpy((unsigned long)inst->description,(unsigned long)"creates a file devive for sim root folder");
			DevLink(&this->DevLink_0);
			if(this->DevLink_0.status != ERR_FUB_BUSY) {
				if(this->DevLink_0.status == ERR_OK) {
					this->DevUnlink_0.handle 	= this->DevLink_0.handle;
					this->DevLink_0.enable 		= false;
					DevLink(&this->DevLink_0);
					this->brdkFileCreateSubFolders_0.enable = true;
					brdkStrCpy((unsigned long)this->brdkFileCreateSubFolders_0.path,(unsigned long)sim->pcRootFolder);
					brdkStrCpy((unsigned long)this->brdkFileCreateSubFolders_0.fileDevice,this->DevLink_0.pDevice);
					brdkFileCreateSubFolders(&this->brdkFileCreateSubFolders_0);
					this->fileState 			= 220;
				}
				else {
					brdkStrCpy((unsigned long)inst->description,(unsigned long)"error calling DevLink. Flip enable to reset fb.");
					inst->status 				= this->DevLink_0.status;
					this->DevLink_0.enable 		= false;
					DevLink(&this->DevLink_0);
					this->fileState 			= 900;
				}
			}
			break;

		case 220:
			brdkStrCpy((unsigned long)inst->description,(unsigned long)"creates the needed folders");
			brdkFileCreateSubFolders(&this->brdkFileCreateSubFolders_0);
			if(this->brdkFileCreateSubFolders_0.done) {
				this->brdkFileCreateSubFolders_0.enable = false;
				brdkFileCreateSubFolders(&this->brdkFileCreateSubFolders_0);
				this->DevUnlink_0.enable 	= true;
				this->fileState				= 230;
			}
			else if(this->brdkFileCreateSubFolders_0.status != ERR_FUB_BUSY) {
				brdkStrCpy((unsigned long)inst->description,(unsigned long)"error calling brdkFileCreateSubFolders. Flip enable to reset fb.");
				inst->status 				= this->brdkFileCreateSubFolders_0.status;
				this->brdkFileCreateSubFolders_0.enable = false;
				brdkFileCreateSubFolders(&this->brdkFileCreateSubFolders_0);
				this->fileState 			= 900;
			}
			break;

		case 230:
			DevUnlink(&this->DevUnlink_0);
			if(this->DevUnlink_0.status != ERR_FUB_BUSY) {
				if(this->DevUnlink_0.status == ERR_OK) {
					this->DevUnlink_0.enable = false;
					DevUnlink(&this->DevUnlink_0);
					this->fileState 			= 0;
				}
				else {
					inst->status 				= this->DevUnlink_0.status;
					this->DevUnlink_0.enable 	= false;
					DevUnlink(&this->DevUnlink_0);
					brdkStrCpy((unsigned long)inst->description,(unsigned long)"error calling DevUnlink. Flip enable to reset fb.");
					this->fileState 			= 900;
				}
			}
			break;

		case 900: /* error state */
			if(!inst->enable) {
				inst->status 	= 0;
				this->fileState = 0;
			}
			break;

	}

}
```

#### brdkFileWrite.c - Write data to a file.
```c
#include <brdkFile_func.h>

void brdkFileWrite(struct brdkFileWrite* inst) {
	brdk_file_write_internal_typ* this = (brdk_file_write_internal_typ*)&inst->internal;

	if(inst->enable) {

		switch(this->state) {

			case 0: /* initialize fb */
					inst->status 				= ERR_FUB_BUSY;
					this->FileCreate_0.enable 	= false;
					FileCreate(&this->FileCreate_0);
					this->FileCreate_0.enable 	= true;
					this->FileCreate_0.pDevice 	= inst->pFileDevice;
					this->FileCreate_0.pFile 	= inst->pFileName;
					this->state 				= 10;
				break;

			case 10: /* create file */
				FileCreate(&this->FileCreate_0);
				switch(this->FileCreate_0.status) {

					case ERR_OK:
						this->FileWrite_0.enable 	= false;
						FileWrite(&this->FileWrite_0);
						this->FileWrite_0.enable 	= true;
						this->FileWrite_0.ident 	= this->FileCreate_0.ident;
						this->FileWrite_0.offset 	= 0;
						this->FileWrite_0.pSrc 		= inst->pData;
						this->FileWrite_0.len 		= inst->dataLength != 0 ? inst->dataLength : brdkStrLen(inst->pData);
						this->state 				= 40;
						break;

					case fiERR_EXIST:
						if(!inst->overwrite) {
							this->FileOpen_0.enable 	= false;
							FileOpen(&this->FileOpen_0);
							this->FileOpen_0.enable 	= true;
							this->FileOpen_0.pDevice 	= inst->pFileDevice;
							this->FileOpen_0.pFile 		= inst->pFileName;
							this->FileOpen_0.mode 		= fiWRITE_ONLY;
							this->state 				= 20;
						}
						else {
							this->FileDelete_0.enable 	= false;
							FileDelete(&this->FileDelete_0);
							this->FileDelete_0.enable 	= true;
							this->FileDelete_0.pDevice 	= inst->pFileDevice;
							this->FileDelete_0.pName 	= inst->pFileName;
							this->state 				= 30;
						}
						break;

					case ERR_FUB_BUSY:
						break;

					default:
						inst->status 				= this->FileCreate_0.status;
						break;

				}
				break;

			case 20: /* file open */
				FileOpen(&this->FileOpen_0);
				switch(this->FileOpen_0.status) {

					case ERR_OK:
						this->FileWrite_0.enable 	= false;
						FileWrite(&this->FileWrite_0);
						this->FileWrite_0.enable 	= true;
						this->FileWrite_0.ident 	= this->FileCreate_0.ident;
						this->FileWrite_0.offset 	= 0;
						this->FileWrite_0.pSrc 		= inst->pData;
						this->FileWrite_0.len 		= inst->dataLength != 0 ? inst->dataLength : brdkStrLen(inst->pData);
						this->state 				= 40;
						break;

					case ERR_FUB_BUSY:
						break;

					default:
						inst->status 				= this->FileOpen_0.status;
						break;

				}
				break;

			case 30:
				FileDelete(&this->FileDelete_0);
				switch(this->FileDelete_0.status) {

					case ERR_OK: case fiERR_FILE_NOT_FOUND:
						this->FileCreate_0.enable 	= false;
						FileCreate(&this->FileCreate_0);
						this->FileCreate_0.enable 	= true;
						this->FileCreate_0.pDevice 	= inst->pFileDevice;
						this->FileCreate_0.pFile 	= inst->pFileName;
						this->state 				= 10;
						break;

					case ERR_FUB_BUSY:
						break;

					default:
						inst->status 				= this->FileDelete_0.status;
						break;

				}
				break;

			case 40:
				FileWrite(&this->FileWrite_0);
				switch(this->FileWrite_0.status) {

					case ERR_OK:
						this->FileClose_0.enable 	= false;
						FileClose(&this->FileClose_0);
						this->FileClose_0.enable 	= true;
						this->FileClose_0.ident 	= this->FileWrite_0.ident;
						this->state 				= 50;
						break;

					case ERR_FUB_BUSY:
						break;

					default:
						inst->status 				= this->FileWrite_0.status;
						break;

				}
				break;

			case 50:
				FileClose(&this->FileClose_0);
				switch(this->FileClose_0.status) {

					case ERR_OK:	case fiERR_FILE_NOT_OPENED:
						inst->status 	= ERR_OK;
						this->state 	= 60;
						break;

					case ERR_FUB_BUSY: break;

					default:
						inst->status 				= this->FileClose_0.status;
						break;

				}
				break;

			case 60:
				break;

		}
	}
	else {
		inst->status = ERR_FUB_ENABLE_FALSE;
		this->state = 0;
	}
}
```

#### brdkFileRead.c - Read data from a file.
```c
#include <brdkFile_func.h>

void brdkFileRead(struct brdkFileRead* inst) {
	brdk_file_read_internal_typ* this = (brdk_file_read_internal_typ*)&inst->internal;

	if(inst->enable) {

		switch(this->state) {

			case 0: /* initialize fb */
				inst->status = ERR_FUB_BUSY;
				this->FileOpen_0.enable 	= false;
				FileOpen(&this->FileOpen_0);
				this->FileOpen_0.enable 	= true;
				this->FileOpen_0.pDevice 	= inst->pFileDevice;
				this->FileOpen_0.pFile 		= inst->pFileName;
				this->FileOpen_0.mode 		= fiREAD_ONLY;
				this->state 				= 10;
				break;

			case 10: /* file open */
				FileOpen(&this->FileOpen_0);
				switch(this->FileOpen_0.status) {

					case ERR_OK:
						if(inst->dataLength >= this->FileOpen_0.filelen+1) {	/* validate that we have enough space to read the file and a 0 */
							brdkStrMemClear(inst->pData,this->FileOpen_0.filelen+1); /* clear enough emeory to read the file */
							this->FileRead_0.enable 	= false;
							FileRead(&this->FileRead_0);
							this->FileRead_0.enable 	= true;
							this->FileRead_0.ident 		= this->FileOpen_0.ident;
							this->FileRead_0.offset 	= 0;
							this->FileRead_0.pDest 		= inst->pData;
							this->FileRead_0.len 		= this->FileOpen_0.filelen;
							this->state 				= 20;
						}
						else {
							inst->status = fiERR_SPACE;
							this->state = 40;
						}
						break;

					case ERR_FUB_BUSY:
						break;

					default:
						inst->status = this->FileOpen_0.status;
						break;

				}
				break;

			case 20: /* read the file */
				FileRead(&this->FileRead_0);
				switch(this->FileRead_0.status) {

					case ERR_OK:
						this->FileClose_0.enable 	= false;
						FileClose(&this->FileClose_0);
						this->FileClose_0.enable 	= true;
						this->FileClose_0.ident 	= this->FileOpen_0.ident;
						this->state 				= 30;
						break;

					case ERR_FUB_BUSY:
						break;

					default:
						inst->status = this->FileRead_0.status;
						break;

				}
				break;

			case 30:
				FileClose(&this->FileClose_0);
				switch(this->FileClose_0.status) {

					case ERR_OK: case fiERR_FILE_NOT_OPENED:
						inst->status				= ERR_OK;
						this->state 				= 40;
						break;

					case ERR_FUB_BUSY:
						break;

					default:
						inst->status = this->FileRead_0.status;
						break;

				}
				break;

			case 40:
				break;

		}
	}
	else {
		inst->status = ERR_FUB_ENABLE_FALSE;
		this->state = 0;
	}
}
```

- CHANGELOG - brdkFile change log file (not shown)

### Library Logical/Libraries/brdkREST (ANSIC, version 1.02.0) - A wrapper library for easy creation of REST clients and servers.
Depends on: AsHttp, brdkSTR, AsARCfg, AsIODiag, brdkJSON

#### brdkREST.typ - Exported data types
```iecst
TYPE
	brdk_rest_response_action_typ :
		( (*Response action type.*)
		BRDK_REST_NO_RESPONSE := 0, (*No response set.*)
		BRDK_REST_200_OK := 200, (*HTTP status 200 OK.*)
		BRDK_REST_400_BAD_REQUEST := 400, (*HTTP status 400 Bad request.*)
		BRDK_REST_401_UNAUTHORIZED := 401, (*HTTP status 401 Unauthorized.*)
		BRDK_REST_403_FORBIDDEN := 403, (*HTTP status 403 Forbidden.*)
		BRDK_REST_404_NOT_FOUND := 404, (*HTTP status 404 Not found.*)
		BRDK_REST_500_INT_SERVER_ERROR := 500, (*HTTP status 500 Internal Server Error.*)
		BRDK_REST_501_NOT_IMPLEMENTED := 501, (*HTTP status 501 Not Implemented.*)
		BRDK_REST_503_SRV_UNAVAILABLE := 503, (*HTTP status 503 Service Unavailable.*)
		BRDK_REST_ABORT := 999 (*Send abort.*)
		);
	brdk_rest_protocol_typ :
		( (*Protocol type.*)
		BRDK_REST_HTTP := 0, (*HTTP protocol.*)
		BRDK_REST_HTTPS := 1 (*HTTPS protocol.*)
		);
	brdk_rest_method_typ :
		( (*Method type.*)
		BRDK_REST_GET := 0, (*Get method.*)
		BRDK_REST_POST := 1, (*Post method.*)
		BRDK_REST_PUT := 2, (*Put method.*)
		BRDK_REST_DELETE := 3 (*Delete method.*)
		);
	brdk_rest_client_internal_typ : 	STRUCT  (*Internal variables.*)
		state : DINT; (*Internal state.*)
		httpsClient_0 : httpsClient; (*httpsClient fb.*)
		httpClient_0 : httpClient; (*httpClient fb.*)
		httpRequestHeader : httpRequestHeader_t; (*httpRequestHeader_t structure.*)
		httpResponseHeader : httpResponseHeader_t; (*httpResponseHeader_t structure.*)
		uri : STRING[BRDK_REST_URI_STRING_MAX_SIZE]; (*URI string.*)
	END_STRUCT;
	brdk_rest_server_request_typ : 	STRUCT  (*Server request type.*)
		header : httpRequestHeader_t; (*Request header.*)
		pQuery : UDINT; (*Pointer to request query data.*)
		maxQuerySize : UDINT; (*Maximum size of query data.*)
		pBody : UDINT; (*Pointer to request body data.*)
		maxBodySize : UDINT; (*Maximum size of body data.*)
	END_STRUCT;
	brdk_rest_server_response_typ : 	STRUCT  (*Server response type.*)
		header : httpResponseHeader_t; (*Response header.*)
		pReponse : UDINT; (*Pointer to reponse data.*)
		length : UDINT; (*Length of reponse data.*)
	END_STRUCT;
	brdk_rest_server_internal_typ : 	STRUCT  (*Internal variables.*)
		state : DINT; (*Internal state.*)
		httpsService_0 : httpsService; (*httpsClient fb.*)
		httpService_0 : httpService; (*httpClient fb.*)
		httpRequestHeader : httpRequestHeader_t; (*httpRequestHeader_t structure.*)
		httpResponseHeader : httpResponseHeader_t; (*httpResponseHeader_t structure.*)
		uri : STRING[BRDK_REST_URI_STRING_MAX_SIZE]; (*URI string.*)
		CfgGetIPAddr_0 : CfgGetIPAddr; (*CfgGetIPAddr fb.*)
	END_STRUCT;
	brdk_rest_content_typ :
		( (*Content types.*)
		BRDK_REST_NONE := 0, (*text/html*)
		BRDK_REST_HTML := 1, (*text/html*)
		BRDK_REST_TEXT := 2, (*text/plain*)
		BRDK_REST_JSON := 3, (*application/json*)
		BRDK_REST_XML := 4, (*application/xml*)
		BRDK_REST_CSV := 5, (*text/csv*)
		BRDK_REST_CSS := 6, (*text/css*)
		BRDK_REST_JAVASCRIPT := 7, (*text/javascript*)
		BRDK_REST_JPEG := 8, (*image/jpeg*)
		BRDK_REST_GZIP := 9, (*application/gzip*)
		BRDK_REST_ZIP := 10, (*application/zip*)
		BRDK_REST_PNG := 11, (*image/png*)
		BRDK_REST_GIF := 12, (*image/gif*)
		BRDK_REST_BMP := 13, (*image/bmp*)
		BRDK_REST_JPG := 14 (*image/jpg*)
		);
	brdk_rest_client_add_to_typ :
		( (*Add to type.*)
		BRDK_REST_PARAMETERS := 0, (*Part of parameter query.*)
		BRDK_REST_HEADER := 1, (*Part of header.*)
		BRDK_REST_BODY_JSON := 2 (*Part of body in JSON format.*)
		);
	brdk_rest_client_params_typ : 	STRUCT  (*Parameters.*)
		addTo : brdk_rest_client_add_to_typ := BRDK_REST_PARAMETERS; (*Add to type.*)
		pKey : UDINT; (*String pointer to key.*)
		pValue : UDINT; (*Pointer to value.*)
		datatype : brdk_json_dt_typ := BRDK_JSON_STRING_TO_STRING; (*Value datatype. Used for sending in JSON body format.*)
	END_STRUCT;
	brdk_rest_server_params_typ : 	STRUCT  (*Parameters.*)
		from : brdk_rest_client_add_to_typ := BRDK_REST_PARAMETERS; (*Add to type.*)
		pKey : UDINT; (*String pointer to key.*)
		pValue : UDINT; (*Pointer to value.*)
		datatype : brdk_json_dt_typ := BRDK_JSON_STRING_TO_STRING; (*Value datatype. Used for sending in JSON body format.*)
	END_STRUCT;
	brdk_rest_imggw_internal_typ : 	STRUCT  (*Internal variables.*)
		state : DINT := 0; (*Internal state.*)
		brdkRESTClient_0 : brdkRESTClient; (*brdkRESTClient.*)
		brdkRESTServer_0 : brdkRESTServer; (*brdkRESTServer.*)
		httpEncodeBase64_0 : httpEncodeBase64; (*httpEncodeBase64_0.*)
		serverState : DINT := 0; (*Internal server state.*)
		length : DINT := 0; (*Data length.*)
	END_STRUCT;
END_TYPE
```

#### brdkREST.var - Exported constants
```iecst
(*SERVER SETTINGS*)
VAR CONSTANT
	BRDK_REST_SERVER_URI_MAX_SIZE : UDINT := 999; (*URI data size. 999 means 1000*)
	BRDK_REST_SERVER_REQ_MAX_SIZE : UDINT := 999; (*Request data size. 999 means 1000*)
	BRDK_REST_SERVER_RES_MAX_SIZE : UDINT := 999; (*Response data size. 999 means 1000*)
	BRDK_REST_URL_MAX_SIZE : UINT := 255; (*Max. size of URL string.*)
	BRDK_REST_PARAMS_MAX_SIZE : UINT := 7; (*7 means 8.*)
	BRDK_REST_URI_STRING_MAX_SIZE : UINT := 499; (*499 means 500.*)
	BRDK_REST_PARAMS_VAL_MAX_SIZE : UINT := 99; (*99 means 100.*)
END_VAR
```

#### brdkREST.fun - Exported functions and function blocks
```iecst
FUNCTION_BLOCK brdkRESTClient (*REST client implementation.*) (*$GROUP=User,$CAT=User,$GROUPICON=User.png,$CATICON=User.png*)
	VAR_INPUT
		enable : BOOL := FALSE; (*Enables the function block.*)
		pURL : UDINT := 0; (*String pointer to host URL.*)
		port : UINT := 0; (*Host port number. Default for http is 80, https is 443.*)
		method : brdk_rest_method_typ := BRDK_REST_GET; (*Method.*)
		contentType : brdk_rest_content_typ := BRDK_REST_HTML; (*Content type.*)
		parameters : ARRAY[0..BRDK_REST_PARAMS_MAX_SIZE] OF brdk_rest_client_params_typ; (*Parameters array.*)
		pRequestBody : UDINT := 0; (*String pointer to request body.*)
		requestBodyLength : UDINT := 0; (*Length of request body. If 0 then string length of pBody is used.*)
		requestBodyMaxSize : UDINT := 0; (*Max size of request body buffer area.*)
		pResponseBody : UDINT := 0; (*String pointer to response data.*)
		responseBodyMaxSize : UDINT := 0; (*Max size of response body buffer area.*)
	END_VAR
	VAR_OUTPUT
		status : UINT := ERR_FUB_ENABLE_FALSE; (*Status of the function block.*)
		responseLength : UDINT := 0; (*Length of reponse data.*)
		responseContentType : brdk_rest_content_typ := BRDK_REST_HTML; (*Response content type.*)
		httpStatus : UINT := 0; (*HTTP status code.*)
	END_VAR
	VAR
		internal : brdk_rest_client_internal_typ; (*Internal variables.*)
	END_VAR
END_FUNCTION_BLOCK

FUNCTION_BLOCK brdkRESTServer (*REST server implementation.*) (*$GROUP=User,$CAT=User,$GROUPICON=User.png,$CATICON=User.png*)
	VAR_INPUT
		enable : BOOL := FALSE; (*Enables the function block.*)
		pName : UDINT := 0; (*String pointer to the name of the service.*)
		protocol : brdk_rest_protocol_typ := BRDK_REST_HTTP; (*Protocol type.*)
		pRequestBody : UDINT := 0; (*String pointer to request body.*)
		requestBodyMaxLength : UDINT := 0; (*Max. length of the request body.*)
		pResponseBody : UDINT := 0; (*String pointer to response data.*)
		responseBodyLength : UDINT := 0; (*Length of response body. If 0 then string length of pBody is used.*)
		responseContentType : brdk_rest_content_typ := BRDK_REST_HTML; (*Response content type.*)
		responseAction : brdk_rest_response_action_typ := BRDK_REST_NO_RESPONSE; (*Response action.*)
		parameters : ARRAY[0..BRDK_REST_PARAMS_MAX_SIZE] OF brdk_rest_server_params_typ; (*Parameters array.*)
	END_VAR
	VAR_OUTPUT
		requestMethod : brdk_rest_method_typ := BRDK_REST_GET; (*Request method.*)
		requestLength : UDINT := 0; (*Length of request data.*)
		requestContentType : brdk_rest_content_typ := BRDK_REST_HTML; (*Request content type.*)
		status : UINT := ERR_FUB_ENABLE_FALSE; (*Status of the function block.*)
		url : STRING[BRDK_REST_URL_MAX_SIZE] := ''; (*REST service URL for easy reading and distribution.*)
	END_VAR
	VAR
		internal : brdk_rest_server_internal_typ; (*Internal variables.*)
	END_VAR
END_FUNCTION_BLOCK

FUNCTION_BLOCK brdkRESTImgGW (*An image gateway. Gets an image from an URL and hosts a 64 based version of the image.*) (*$GROUP=User,$CAT=User,$GROUPICON=User.png,$CATICON=User.png*)
	VAR_INPUT
		enable : BOOL := FALSE; (*Enables the function block.*)
		pURL : UDINT := 0; (*String pointer for the URL for the image.*)
		port : UINT := 0; (*Host port number. Default for http is 80, https is 443.*)
		pRawImgBuffer : UDINT := 0; (*Data buffer for the raw image.*)
		rawImgBufferSize : UDINT := 0; (*Size of the raw image buffer area.*)
		pName : UDINT := 0; (*String pointer to the name of the service.*)
		protocol : brdk_rest_protocol_typ := BRDK_REST_HTTP; (*Protocol type.*)
		parameters : ARRAY[0..BRDK_REST_PARAMS_MAX_SIZE] OF brdk_rest_client_params_typ; (*Parameters array.*)
		pEncodedImgBuffer : UDINT := 0; (*Data buffer for the encoded image.*)
		encodedImgBufferSize : UDINT := 0; (*Size of the encoded image buffer area.*)
	END_VAR
	VAR_OUTPUT
		status : UINT := ERR_FUB_ENABLE_FALSE; (*Status of the function block.*)
	END_VAR
	VAR
		internal : brdk_rest_imggw_internal_typ; (*Internal variables.*)
	END_VAR
END_FUNCTION_BLOCK
```

#### brdkRESTClient.c - brdkRESTClient implementation.
```c
#include <brdkREST_func.h>

void brdkRESTClient(struct brdkRESTClient* inst) {
	brdk_rest_client_internal_typ* this = (brdk_rest_client_internal_typ*)&inst->internal;
	signed long startPos;
	unsigned long i, j, init;
	unsigned char questionAdded;

	if(inst->enable) {

		switch(this->state) {

			case 0:	/* setup httpClient fb */
				inst->status 			= ERR_FUB_BUSY;
				inst->httpStatus 		= 0;
				inst->responseLength 	= 0;
				startPos = brdkStrSearch(inst->pURL,(unsigned long)&"://");
				if(startPos > -1) startPos += 3;
				else startPos = 0;

				i = 0;
				brdkStrCpy((unsigned long)&this->uri,(unsigned long)&"");
				brdkStrMemClear((unsigned long)&this->httpRequestHeader.host,sizeof(this->httpRequestHeader.host));
				while(((char*)inst->pURL)[startPos] != BRDK_STR_ASCII_FRONT_SLASH && ((char*)inst->pURL)[startPos] != BRDK_STR_ASCII_NULL) {
					((char*)this->httpRequestHeader.host)[i++] = ((char*)inst->pURL)[startPos++];
				}
				((char*)this->httpRequestHeader.host)[i] = BRDK_STR_ASCII_NULL;
				i = 0;
				while(((char*)inst->pURL)[startPos] != BRDK_STR_ASCII_NULL) {
					this->uri[i++] = ((char*)inst->pURL)[startPos++];
				}
				this->uri[i] = BRDK_STR_ASCII_NULL;

				/* setup request header */
				brdkStrCpy((unsigned long)&this->httpRequestHeader.protocol,(unsigned long)&"HTTP/1.1");
				brdkStrCpy((unsigned long)&this->httpRequestHeader.connection,(unsigned long)&"keep-alive");
				setContentType((unsigned long)&this->httpRequestHeader.contentType, inst->contentType);

				questionAdded = false;
				j = 0;
				init = true;
				startPos = 0;
				for(i = 0; i <= BRDK_REST_PARAMS_MAX_SIZE; i++) {
					if(inst->parameters[i].pKey != 0) {
						switch(inst->parameters[i].addTo) {

							case BRDK_REST_PARAMETERS:
								if(!questionAdded) {
									questionAdded = true;
									brdkStrCat((unsigned long)&this->uri,(unsigned long)&"?");
								}
								else brdkStrCat((unsigned long)&this->uri,(unsigned long)&"&");
								brdkStrCat((unsigned long)&this->uri, inst->parameters[i].pKey);
								brdkStrCat((unsigned long)&this->uri,(unsigned long)&"=");
								brdkStrCat((unsigned long)&this->uri, inst->parameters[i].pValue);
								break;

							case BRDK_REST_HEADER:
								brdkStrCpy((unsigned long)&this->httpRequestHeader.userLine[j].name, inst->parameters[i].pKey);
								brdkStrCpy((unsigned long)&this->httpRequestHeader.userLine[j++].value, inst->parameters[i].pValue);
								break;

							case BRDK_REST_BODY_JSON:
								if(inst->pRequestBody != 0 && inst->requestBodyMaxSize > 0) {
									if(init) {
										init = false;
										brdkStrMemClear(inst->pRequestBody,inst->requestBodyMaxSize);
									}
									startPos = brdkJSONstringify(inst->pRequestBody, inst->parameters[i].pKey, inst->parameters[i].pValue, inst->parameters[i].datatype, inst->requestBodyMaxSize, startPos);
								}
								else {
									inst->status = httpERR_BUFFER_SIZE;
									this->state = 999;
								}
								break;

						}

					}
					else break;
				}
				if(this->state != 999) {
					if(((char*)inst->pURL)[4] == BRDK_STR_ASCII_s) { /* https */
						this->httpsClient_0.enable 				= false;
						httpsClient(&this->httpsClient_0);
						this->httpsClient_0.enable 				= true;
						this->httpsClient_0.pRequestHeader 		= (unsigned long)&this->httpRequestHeader;
						this->httpsClient_0.pResponseHeader 	= (unsigned long)&this->httpResponseHeader;
						this->httpsClient_0.pRequestData		= inst->pRequestBody;
						if(inst->requestBodyLength == 0 && this->httpsClient_0.pRequestData != 0) this->httpsClient_0.requestDataLen = brdkStrLen(this->httpsClient_0.pRequestData);
						else this->httpsClient_0.requestDataLen = inst->requestBodyLength;
						this->httpRequestHeader.contentLength 	= this->httpsClient_0.requestDataLen;
						this->httpsClient_0.pResponseData		= inst->pResponseBody;
						this->httpsClient_0.responseDataSize 	= inst->responseBodyMaxSize;
						this->httpsClient_0.pHost	 			= (unsigned long)&this->httpRequestHeader.host;
						this->httpsClient_0.pUri				= (unsigned long)&this->uri;

						this->httpsClient_0.option 				= httpOPTION_HTTP_11;	/* always use HTTP/1.1 */
						this->httpsClient_0.method				= getMethod(inst->method);
						this->httpsClient_0.send 				= true;
						this->state								= 200;
					}
					else {	/* http */
						this->httpClient_0.enable 			= false;
						httpClient(&this->httpClient_0);
						this->httpClient_0.enable 			= true;
						this->httpClient_0.pRequestHeader 	= (unsigned long)&this->httpRequestHeader;
						this->httpClient_0.pResponseHeader 	= (unsigned long)&this->httpResponseHeader;
						this->httpClient_0.pRequestData		= inst->pRequestBody;
						if(inst->requestBodyLength == 0 && this->httpClient_0.pRequestData != 0) this->httpClient_0.requestDataLen = brdkStrLen(this->httpClient_0.pRequestData);
						else this->httpClient_0.requestDataLen = inst->requestBodyLength;
						this->httpRequestHeader.contentLength 	= this->httpClient_0.requestDataLen;
						this->httpClient_0.pResponseData	= inst->pResponseBody;
						this->httpClient_0.responseDataSize = inst->responseBodyMaxSize;
						this->httpClient_0.pHost 			= (unsigned long)&this->httpRequestHeader.host;
						this->httpClient_0.hostPort 		= inst->port;
						this->httpClient_0.pUri				= (unsigned long)&this->uri;
						this->httpClient_0.option 			= httpOPTION_HTTP_11;	/* always use HTTP/1.1 */
						this->httpClient_0.method			= getMethod(inst->method);
						this->httpClient_0.send 			= true;
						this->state							= 100;
					}
				}
				break;

			case 100:	/* http */
				httpClient(&this->httpClient_0);
				switch(this->httpClient_0.status) {

					case ERR_OK:
						inst->status 				= ERR_OK;
						inst->httpStatus 			= this->httpClient_0.httpStatus;
						inst->responseLength 		= this->httpClient_0.responseDataLen;
						inst->responseContentType 	= findContentType((unsigned long)&this->httpResponseHeader.contentType);
						this->state 				= 300;
						break;

					case ERR_FUB_BUSY:
						break;

					default:
						inst->status = this->httpsClient_0.status;
						this->state = 999;
						break;

				}
				break;

			case 200:	/* https */
				httpsClient(&this->httpsClient_0);
				switch(this->httpsClient_0.status) {

					case ERR_OK:
						inst->status 				= ERR_OK;
						inst->httpStatus 			= this->httpsClient_0.httpStatus;
						inst->responseLength 		= this->httpsClient_0.responseDataLen;
						inst->responseContentType 	= findContentType((unsigned long)&this->httpResponseHeader.contentType);
						this->state 				= 300;
						break;

					case ERR_FUB_BUSY:
						break;

					default:
						inst->status = this->httpsClient_0.status;
						this->state = 999;
						break;

				}
				break;

			case 300: /* done - flip enable to make a new request */
				break;

			case 999: /* error */
				break;

		}

	}
	else {
		switch(this->state) {

			case 100: /* http */
				this->httpClient_0.abort = true;
				httpClient(&this->httpClient_0);
				this->httpClient_0.enable = false;
				httpClient(&this->httpClient_0);
				this->state = 0;
				break;

			case 200: /* https */
				this->httpsClient_0.abort = true;
				httpsClient(&this->httpsClient_0);
				this->httpsClient_0.enable = false;
				httpsClient(&this->httpsClient_0);
				this->state = 0;
				break;

			default:
				this->state = 0;
				inst->status = ERR_FUB_ENABLE_FALSE;

		}
	}
}
```

#### brdkRESTServer.c - brdkRESTServer implementation.
```c
#include <brdkREST_func.h>

void brdkRESTServer(struct brdkRESTServer* inst) {
	brdk_rest_server_internal_typ* this = (brdk_rest_server_internal_typ*)&inst->internal;
	unsigned long i,j;
	unsigned char urlStart;

	if(inst->enable) {
		switch(this->state) {

			case 0:
				inst->status = ERR_FUB_BUSY;
				brdkStrMemClear((unsigned long)&inst->url, sizeof(inst->url));
				brdkStrCpy((unsigned long)&inst->url, (unsigned long)&"http");
				if(inst->protocol != BRDK_REST_HTTP) {
					brdkStrCat((unsigned long)&inst->url, (unsigned long)&"s://");
					urlStart 							= 8;
				}
				else {
					brdkStrCat((unsigned long)&inst->url, (unsigned long)&"://");
					urlStart 							= 7;
				}
				this->CfgGetIPAddr_0.enable 	= false;
				CfgGetIPAddr(&this->CfgGetIPAddr_0);
				this->CfgGetIPAddr_0.enable 	= true;
				this->CfgGetIPAddr_0.pIPAddr 	= (unsigned long)&inst->url[urlStart];
				if(!DiagCpuIsSimulated()) this->CfgGetIPAddr_0.pDevice	= (unsigned long)&"IF3";
				else this->CfgGetIPAddr_0.pDevice	= (unsigned long)&"IF2";
				this->CfgGetIPAddr_0.Len 		= 16;
				this->state						= 10;
				break;

			case 10:
				brdkStrCat((unsigned long)&inst->url, (unsigned long)&"192.168.2.11");
				this->state = 20;
				break;

		/*	case 10:
				CfgGetIPAddr(&this->CfgGetIPAddr_0);
				switch(this->CfgGetIPAddr_0.status) {

					case ERR_OK:
						this->state = 20;
						break;

					case ERR_FUB_BUSY:
						break;

					default:
						if(DiagCpuIsSimulated()) {
							if(inst->protocol != BRDK_REST_HTTP) brdkStrCpy((unsigned long)&inst->url, (unsigned long)&"https://127.0.0.1");
							else brdkStrCpy((unsigned long)&inst->url, (unsigned long)&"http://127.0.0.1");
						}
						this->state = 20;
						break;

				}
				break;
			*/

			case 20:
				brdkStrCat((unsigned long)&inst->url, (unsigned long)&"/");
				brdkStrCat((unsigned long)&inst->url, inst->pName);
				if(inst->protocol != BRDK_REST_HTTP) {
					this->httpsService_0.enable 			= false;
					httpsService(&this->httpsService_0);
					this->httpsService_0.enable 			= true;
					this->httpsService_0.send 				= false;
					this->httpsService_0.abort 				= false;
					this->httpsService_0.option 			= httpOPTION_HTTP_11 + httpOPTION_SERVICE_TYPE_NAME;;
					this->httpsService_0.pServiceName 		= inst->pName;
					this->httpsService_0.pUri 				= (unsigned long)&this->uri;
					this->httpsService_0.uriSize 			= sizeof(this->uri);
					this->httpsService_0.pRequestHeader 	= (unsigned long)&this->httpRequestHeader;
					this->httpsService_0.pRequestData 		= inst->pRequestBody;
					this->httpsService_0.requestDataSize 	= inst->requestBodyMaxLength;
					this->httpsService_0.pResponseHeader 	= (unsigned long)&this->httpResponseHeader;
					this->httpsService_0.pResponseData 		= inst->pResponseBody;
					if(inst->responseBodyLength == 0 && this->httpsService_0.pResponseData != 0) this->httpsService_0.responseDataLen = brdkStrLen(this->httpsService_0.pResponseData);
					else this->httpsService_0.responseDataLen = inst->responseBodyLength;
					this->state								= 200;
				}
				else {
					this->httpService_0.enable 			= false;
					httpService(&this->httpService_0);
					this->httpService_0.enable 			= true;
					this->httpService_0.send 			= false;
					this->httpService_0.abort 			= false;
					this->httpService_0.option 			= httpOPTION_HTTP_11 + httpOPTION_SERVICE_TYPE_NAME;
					this->httpService_0.pServiceName 	= inst->pName;
					this->httpService_0.pUri 			= (unsigned long)&this->uri;
					this->httpService_0.uriSize			= sizeof(this->uri);
					this->httpService_0.pRequestHeader 	= (unsigned long)&this->httpRequestHeader;
					this->httpService_0.pRequestData 	= inst->pRequestBody;
					this->httpService_0.requestDataSize = inst->requestBodyMaxLength;
					this->httpService_0.pResponseHeader = (unsigned long)&this->httpResponseHeader;
					this->httpService_0.pResponseData 	= inst->pResponseBody;
					if(inst->responseBodyLength == 0 && this->httpService_0.pResponseData != 0) this->httpService_0.responseDataLen = brdkStrLen(this->httpService_0.pResponseData);
					else this->httpService_0.responseDataLen = inst->responseBodyLength;
					this->state							= 100;
				}
				j = 0;
				for(i=0; i <= BRDK_REST_PARAMS_MAX_SIZE; i++) {
					if(inst->parameters[i].pKey != 0 && inst->parameters[i].from == BRDK_REST_HEADER) {
						brdkStrCpy((unsigned long)&this->httpRequestHeader.userLine[j++].name, inst->parameters[i].pKey);
					}
				}
				break;

			/* HTTP */
			case 100: /* WAITING FOR INCOMMING CALL */
				this->httpService_0.pResponseData 	= inst->pResponseBody;
				if(inst->responseBodyLength == 0 && this->httpService_0.pResponseData != 0) this->httpService_0.responseDataLen = brdkStrLen(this->httpService_0.pResponseData);
				else this->httpService_0.responseDataLen = inst->responseBodyLength;
				httpService(&this->httpService_0);
				switch(this->httpService_0.status) {

					case ERR_OK:
						switch(this->httpService_0.phase) {

							case httpPHASE_RECEIVED:
								if(!validateServerParams(inst, this)) {
									setHttpStatus(BRDK_REST_400_BAD_REQUEST, (unsigned long)&this->httpResponseHeader.status);
									this->httpService_0.send = true;
								}
								else {
									inst->status = ERR_OK;
									this->state = 300;
								}
								break;

							default:
								this->httpService_0.send = false;
								break;

						}
						break;

					case ERR_FUB_BUSY:
						break;

					default:
						inst->status = this->httpService_0.status;
						this->state = 999;
						break;

				}
				break;

			/* HTTPS */
			case 200: /* WAITING FOR INCOMMING CALL */
				this->httpsService_0.pResponseData 		= inst->pResponseBody;
				if(inst->responseBodyLength == 0 && this->httpsService_0.pResponseData != 0) this->httpsService_0.responseDataLen = brdkStrLen(this->httpsService_0.pResponseData);
				else this->httpsService_0.responseDataLen = inst->responseBodyLength;
				httpsService(&this->httpsService_0);
				switch(this->httpsService_0.status) {

					case ERR_OK:
						switch(this->httpsService_0.phase) {

							case httpPHASE_RECEIVED:
								if(!validateServerParams(inst, this)) {
									setHttpStatus(BRDK_REST_400_BAD_REQUEST, (unsigned long)&this->httpResponseHeader.status);
									this->httpsService_0.send = true;
								}
								else {
									inst->status = ERR_OK;
									this->state = 300;
								}
								break;

							default:
								this->httpsService_0.send = false;
								break;

						}
						break;

					case ERR_FUB_BUSY:
						break;

					default:
						inst->status = this->httpsService_0.status;
						this->state = 999;
						break;

				}
				break;

			/* waiting to send back reply */
			case 300:
				switch(inst->responseAction) {

					case BRDK_REST_NO_RESPONSE:
						break;

					case BRDK_REST_ABORT:
						inst->status = ERR_FUB_BUSY;
						if(inst->protocol != BRDK_REST_HTTP) {
							this->httpsService_0.abort = true;
							this->state = 200;
						}
						else {
							this->httpService_0.abort = true;
							this->state = 100;
						}
						break;

					default:
						inst->status = ERR_FUB_BUSY;
						brdkStrCpy((unsigned long)&this->httpResponseHeader.protocol,(unsigned long)&"HTTP/1.1");
						brdkStrCpy((unsigned long)&this->httpResponseHeader.connection,(unsigned long)&"keep-alive");
						setContentType((unsigned long)&this->httpResponseHeader.contentType, inst->responseContentType);
						setHttpStatus(inst->responseAction, (unsigned long)&this->httpResponseHeader.status);

						if(inst->protocol != BRDK_REST_HTTP) {
							if(inst->responseBodyLength == 0 && this->httpsService_0.pResponseData != 0) this->httpsService_0.responseDataLen = brdkStrLen(this->httpsService_0.pResponseData);
							else this->httpsService_0.responseDataLen = inst->responseBodyLength;
							this->httpResponseHeader.contentLength 	= this->httpsService_0.responseDataLen;

							this->httpsService_0.send = true;
							this->state = 200;

						}
						else {
							if(inst->responseBodyLength == 0 && this->httpService_0.pResponseData != 0) this->httpService_0.responseDataLen = brdkStrLen(this->httpService_0.pResponseData);
							else this->httpService_0.responseDataLen = inst->responseBodyLength;
							this->httpResponseHeader.contentLength 	= this->httpService_0.responseDataLen;

							this->httpService_0.send = true;
							this->state = 100;
						}
						inst->responseAction = BRDK_REST_NO_RESPONSE;
						break;

				}
				break;

			case 999: /* error */
				break;

		}
	}
	else {
		switch(this->state) {

			case 100: /* http */
				this->httpService_0.abort = true;
				httpService(&this->httpService_0);
				this->httpService_0.enable = false;
				httpService(&this->httpService_0);
				this->state = 0;
				break;

			case 200: /* https */
				this->httpsService_0.abort = true;
				httpsService(&this->httpsService_0);
				this->httpsService_0.enable = false;
				httpsService(&this->httpsService_0);
				this->state = 0;
				break;

			default:
				this->state = 0;
				inst->status = ERR_FUB_ENABLE_FALSE;

		}
	}

}
```

#### brdkRESTImgGW.c - brdkRESTImgGW implementation.
```c
#include <brdkREST_func.h>

void brdkRESTImgGW(struct brdkRESTImgGW* inst) {
	brdk_rest_imggw_internal_typ* this = (brdk_rest_imggw_internal_typ*)&inst->internal;

	if(inst->enable) {

		switch(this->state) {

			case 0: /* prepare the http client call */
				inst->status = ERR_FUB_BUSY;
				brdkStrMemClear(inst->pRawImgBuffer,inst->rawImgBufferSize);
				this->brdkRESTClient_0.enable 				= false;
				brdkRESTClient(&this->brdkRESTClient_0);
				this->brdkRESTClient_0.enable 				= true;
				this->brdkRESTClient_0.pURL 				= inst->pURL;
				this->brdkRESTClient_0.port 				= inst->port;
				this->brdkRESTClient_0.pResponseBody 		= inst->pRawImgBuffer;
				this->brdkRESTClient_0.responseBodyMaxSize 	= inst->rawImgBufferSize;
				brdkStrMemCpy((unsigned long)&this->brdkRESTClient_0.parameters,(unsigned long)&inst->parameters,sizeof(inst->parameters));
				this->state 								= 10;
				break;

			case 10: /* request for the image */
				brdkRESTClient(&this->brdkRESTClient_0);
				switch(this->brdkRESTClient_0.status) {

					case ERR_OK:
						brdkStrMemClear(inst->pEncodedImgBuffer,inst->encodedImgBufferSize);
						brdkStrCpy(inst->pEncodedImgBuffer,(unsigned long)&"<img src=\"data:image/");
						switch(this->brdkRESTClient_0.responseContentType) {
							case BRDK_REST_JPEG: brdkStrCat(inst->pEncodedImgBuffer,(unsigned long)&"jpeg"); break;
							case BRDK_REST_PNG: brdkStrCat(inst->pEncodedImgBuffer,(unsigned long)&"png"); break;
							case BRDK_REST_GIF: brdkStrCat(inst->pEncodedImgBuffer,(unsigned long)&"gif"); break;
							case BRDK_REST_BMP: brdkStrCat(inst->pEncodedImgBuffer,(unsigned long)&"bmp"); break;
							default: brdkStrCat(inst->pEncodedImgBuffer,(unsigned long)&"jpg"); break;

						}
						brdkStrCat(inst->pEncodedImgBuffer,(unsigned long)&";base64,");
						this->httpEncodeBase64_0.enable 	= true;
						this->httpEncodeBase64_0.pSrc 		= this->brdkRESTClient_0.pResponseBody;
						this->httpEncodeBase64_0.srcLen 	= this->brdkRESTClient_0.responseLength;
						this->length 						= brdkStrLen(inst->pEncodedImgBuffer);
						this->httpEncodeBase64_0.pDest 		= inst->pEncodedImgBuffer+this->length;
						this->httpEncodeBase64_0.destSize 	= inst->encodedImgBufferSize-this->length;
						this->state 						= 20;
						break;

					case ERR_FUB_BUSY:
						break;

					default:
						inst->status = this->brdkRESTClient_0.status;
						this->state = 999;
						break;

				}
				break;

			case 20: /* encode the raw image to base 64 */
				httpEncodeBase64(&this->httpEncodeBase64_0);
				switch(this->httpEncodeBase64_0.status) {

					case ERR_OK:
						brdkStrCat(inst->pEncodedImgBuffer,(unsigned long)&"\">");
						this->length += this->httpEncodeBase64_0.destLen + 2;
						inst->status = ERR_OK;
						this->state = 30;
						break;

					case ERR_FUB_BUSY:
						break;

					default:
						inst->status = this->httpEncodeBase64_0.status;
						this->state = 999;
						break;

				}
				break;

		}

		/* server state machine */
		switch(this->serverState) {

			case 0: /* prepare the server */
				this->brdkRESTServer_0.enable 				= true;
				this->brdkRESTServer_0.pName 				= inst->pName;
				this->brdkRESTServer_0.protocol 			= inst->protocol;
				this->brdkRESTServer_0.responseContentType 	= BRDK_REST_HTML;
				this->serverState 								= 10;
				break;

			case 10: /* wait for the call */
				switch(this->brdkRESTServer_0.status) {

					case ERR_OK:
						switch(this->state) {

							case 30:
								this->brdkRESTServer_0.pResponseBody 		= inst->pEncodedImgBuffer;
								this->brdkRESTServer_0.responseBodyLength 	= this->length;
								this->brdkRESTServer_0.responseAction 		= BRDK_REST_200_OK;
								break;

							default:
								this->brdkRESTServer_0.pResponseBody 		= 0;
								this->brdkRESTServer_0.responseBodyLength 	= 0;
								this->brdkRESTServer_0.responseAction 		= BRDK_REST_503_SRV_UNAVAILABLE;
								break;

						}

						break;

					case ERR_FUB_BUSY:
						break;

					default:
						inst->status = this->brdkRESTServer_0.status;
						this->serverState = 999;
						this->state = 999;
						break;

				}
				break;

		}
		brdkRESTServer(&this->brdkRESTServer_0);

	}
	else {
		inst->status 					= ERR_FUB_ENABLE_FALSE;
		this->state 					= 0;
		this->serverState 				= 0;
		this->brdkRESTServer_0.enable 	= false;
		brdkRESTServer(&this->brdkRESTServer_0);
		this->brdkRESTClient_0.enable 	= false;
		brdkRESTClient(&this->brdkRESTClient_0);
	}
}
```

#### brdkREST_func.h - Header for internal functions for library.
```c
#ifndef BRDK_REST_FUNCS
#define BRDK_REST_FUNCS 1

#include <brdkREST.h>
#include <bur/plctypes.h>

#ifdef __cplusplus
	extern "C"
	{
#endif

#ifdef __cplusplus
	};
#endif

#define false 0
#define true 1
#define NULL 0

unsigned short getMethod(brdk_rest_method_typ method);
brdk_rest_method_typ setMethod(unsigned short method);
brdk_rest_content_typ findContentType(unsigned long pStr);
void setContentType(unsigned long pDestination, brdk_rest_content_typ type);
void setHttpStatus(brdk_rest_response_action_typ status, unsigned long pStr);
unsigned char validateServerParams(brdkRESTServer_typ* inst, brdk_rest_server_internal_typ* this);

#endif /* !BRDK_REST_FUNCS */
```
